# B&R Automation Studio project ControlPLC_DataDistribution (part 6)

#### vfAddAlarm.c
```c
#include <bur/plctypes.h>
#ifdef __cplusplus
	extern "C"
	{
#endif
	#include "VFAlarms.h"
#ifdef __cplusplus
	};
#endif
#include "string.h"

/* TODO: Add your comment here */
plcbit vfAddAlarm(plcstring* name, plcstring* scope, unsigned long code, enum vfALARMS_SEVERITY_enum severity, enum vfALARMS_BEHAVIOR_enum behavior, struct vfAlarms_Data_typ* data)
{

	vfAddAlarmTextScope( name, scope, "", code, severity, behavior, data);

	return 1;
}

plcbit vfAddAlarmApi(struct vfAlarms_Instance_type* name, plcstring* scope, unsigned long code, enum vfALARMS_SEVERITY_enum severity, enum vfALARMS_BEHAVIOR_enum behavior, struct vfAlarms_Data_typ* data){

	vfAddAlarm(name->_,  scope, code, severity, behavior, data);

	STRING snippet[vfALARMS_MAX_SNIPPET_PV_NAME_LEN];
	stringlcpy( snippet, data->in.snippetPvName, vfALARMS_MAX_SNIPPET_PV_NAME_LEN);
	stringlcat( snippet, ".", vfALARMS_MAX_SNIPPET_PV_NAME_LEN);
	stringlcat( snippet, name->snippet, vfALARMS_MAX_SNIPPET_PV_NAME_LEN);

	vfAddSnippet( name->snippet, snippet, data);

}

/* TODO: Add your comment here */
plcbit vfAddAlarmTextScope(plcstring* name, plcstring* scope, plcstring* textScope, unsigned long code, enum vfALARMS_SEVERITY_enum severity, enum vfALARMS_BEHAVIOR_enum behavior, struct vfAlarms_Data_typ* data)
{
	// Error check inputs.
	if (!data) return 0;
	if (!name) return 0;

	// Look for first empty spot, and add new alarm info there.
	int i;
	for (i = 0; i < vfALARMS_MAX_ALARMS; i++) {
		if (!strcmp(data->internal.alarms[i].name, "")) {
			// Found an empty location. Add our string.
			strcpy(data->internal.alarms[i].name, name);
			if (!strcmp(scope, "")) {
				strcpy(data->internal.alarms[i].scope, data->in.scope);
			} else {
				strcpy(data->internal.alarms[i].scope, scope);
			}

			if (!strcmp(textScope, "")) {
				strcpy(data->internal.alarms[i].textScope, data->in.scope);
			} else{
				strcpy(data->internal.alarms[i].textScope, textScope);
			}
			data->internal.alarms[i].code = code;
			data->internal.alarms[i].severity = severity;
			data->internal.alarms[i].behavior = behavior;
			break;
		}
	}

	return 1;
}

plcbit vfAddAlarmTextScopeApi(struct vfAlarms_Instance_type* name, plcstring* scope, plcstring* textScope, unsigned long code, enum vfALARMS_SEVERITY_enum severity, enum vfALARMS_BEHAVIOR_enum behavior, struct vfAlarms_Data_typ* data){

	vfAddAlarmTextScope(name->_,  scope, textScope, code, severity, behavior, data);

	STRING snippet[vfALARMS_MAX_SNIPPET_PV_NAME_LEN];
	stringlcpy( snippet, data->in.snippetPvName, vfALARMS_MAX_SNIPPET_PV_NAME_LEN);
	stringlcat( snippet, ".", vfALARMS_MAX_SNIPPET_PV_NAME_LEN);
	stringlcat( snippet, name->snippet, vfALARMS_MAX_SNIPPET_PV_NAME_LEN);

	vfAddSnippet( name->snippet, snippet, data);

}
```

#### vfAddSnippet.c
```c
#include <bur/plctypes.h>
#ifdef __cplusplus
	extern "C"
	{
#endif
	#include "VFAlarms.h"
#ifdef __cplusplus
	};
#endif
#include "string.h"

/* TODO: Add your comment here */
plcbit vfAddSnippet(plcstring* key, plcstring* pvName, struct vfAlarms_Data_typ* data)
{
	// Error check inputs.
	if (!data) return 0;
	if (!key) return 0;
	if (!pvName) return 0;

	// Look for first empty spot, and add new snippet info there.
	int i;
	for (i = 0; i < vfALARMS_MAX_SNIPPETS; i++) {
		if (!strcmp(data->internal.snippets[i].key, "")) {
			// Found an empty location. Add our string.
			strcpy(data->internal.snippets[i].key, key);
			strcpy(data->internal.snippets[i].pvName, pvName);
			break;
		}
	}

	return 1;
}
```

#### vfAddReactionByName.c
```c
#include <bur/plctypes.h>
#ifdef __cplusplus
	extern "C"
	{
#endif
	#include "VFAlarms.h"
#ifdef __cplusplus
	};
#endif
#include "string.h"

/* TODO: Add your comment here */
plcbit vfAddReactionByName(plcstring* name, plcstring* reactionName1, plcstring* reactionName2, plcstring* reactionName3, plcstring* reactionName4, plcstring* reactionName5, plcstring* reactionName6, struct vfAlarms_Data_typ* data)
{
	// Error check inputs.
	if (!data) return 0;
	if (!name) return 0;

	// Look for first empty spot, and add new alarm info there.
	int i;
	for (i = 0; i < vfALARMS_MAX_MAPPINGS; i++) {
		if (!strcmp(data->internal.reactions.byName[i].name, "")) {
			// Found an empty location. Add our info.
			strcpy(data->internal.reactions.byName[i].name, name);
			strcpy(data->internal.reactions.byName[i].reactionName[0], reactionName1);
			strcpy(data->internal.reactions.byName[i].reactionName[1], reactionName2);
			strcpy(data->internal.reactions.byName[i].reactionName[2], reactionName3);
			strcpy(data->internal.reactions.byName[i].reactionName[3], reactionName4);
			strcpy(data->internal.reactions.byName[i].reactionName[4], reactionName5);
			strcpy(data->internal.reactions.byName[i].reactionName[5], reactionName6);
			break;
		}
	}

	return 1;
}
```

#### vfAddReactionBySeverity.c
```c
#include <bur/plctypes.h>
#ifdef __cplusplus
	extern "C"
	{
#endif
	#include "VFAlarms.h"
#ifdef __cplusplus
	};
#endif
#include "string.h"

/* TODO: Add your comment here */
plcbit vfAddReactionBySeverity(enum vfALARMS_SEVERITY_enum severity, plcstring* reactionName1, plcstring* reactionName2, plcstring* reactionName3, plcstring* reactionName4, plcstring* reactionName5, plcstring* reactionName6, struct vfAlarms_Data_typ* data)
{
	// Error check inputs.
	if (!data) return 0;

	// Look for first empty spot, and add new alarm info there.
	int i;
	for (i = 0; i < vfALARMS_MAX_MAPPINGS; i++) {
		if (data->internal.reactions.bySeverity[i].severity == vfALARMS_SEVERITY_NONE) {
			// Found an empty location. Add our info.
			data->internal.reactions.bySeverity[i].severity = severity;
			strcpy(data->internal.reactions.bySeverity[i].reactionName[0], reactionName1);
			strcpy(data->internal.reactions.bySeverity[i].reactionName[1], reactionName2);
			strcpy(data->internal.reactions.bySeverity[i].reactionName[2], reactionName3);
			strcpy(data->internal.reactions.bySeverity[i].reactionName[3], reactionName4);
			strcpy(data->internal.reactions.bySeverity[i].reactionName[4], reactionName5);
			strcpy(data->internal.reactions.bySeverity[i].reactionName[5], reactionName6);
			break;
		}
	}

	return 1;
}
```

#### vfAddAggregationByName.c
```c
#include <bur/plctypes.h>
#ifdef __cplusplus
	extern "C"
	{
#endif
	#include "VFAlarms.h"
#ifdef __cplusplus
	};
#endif
#include "string.h"

/* TODO: Add your comment here */
plcbit vfAddAggregationByName(plcstring* name, plcstring* aggregationName, struct vfAlarms_Data_typ* data)
{
	// Error check inputs.
	if (!data) return 0;
	if (!name) return 0;

	// Look for first empty spot, and add new alarm info there.
	int i;
	for (i = 0; i < vfALARMS_MAX_MAPPINGS; i++) {
		if (!strcmp(data->internal.aggregations.byName[i].name, "")) {
			// Found an empty location. Add our info.
			strcpy(data->internal.aggregations.byName[i].name, name);
			strcpy(data->internal.aggregations.byName[i].aggregationName, aggregationName);
			break;
		}
	}

	return 1;
}

plcbit vfAddAggregationByNameApi(plcstring* name, struct vfAlarms_Instance_type* aggregationName, struct vfAlarms_Data_typ* data){

	vfAddAggregationByName( name, aggregationName->_, data);

}
```

#### vfAddAggregationBySeverity.c
```c
#include <bur/plctypes.h>
#ifdef __cplusplus
	extern "C"
	{
#endif
	#include "VFAlarms.h"
#ifdef __cplusplus
	};
#endif
#include "string.h"

/* TODO: Add your comment here */
plcbit vfAddAggregationBySeverity(enum vfALARMS_SEVERITY_enum severity, plcstring* aggregationName, struct vfAlarms_Data_typ* data)
{
	// Error check inputs.
	if (!data) return 0;

	// Look for first empty spot, and add new alarm info there.
	int i;
	for (i = 0; i < vfALARMS_MAX_MAPPINGS; i++) {
		if (data->internal.aggregations.bySeverity[i].severity == vfALARMS_SEVERITY_NONE) {
			// Found an empty location. Add our info.
			data->internal.aggregations.bySeverity[i].severity = severity;
			strcpy(data->internal.aggregations.bySeverity[i].aggregationName, aggregationName);
			break;
		}
	}

	return 1;
}
```

#### vfSetDefaultMapping.c
```c
#include <bur/plctypes.h>
#ifdef __cplusplus
	extern "C"
	{
#endif
	#include "VFAlarms.h"
#ifdef __cplusplus
	};
#endif
#include "string.h"

/* TODO: Add your comment here */
plcbit vfSetDefaultMapping(enum vfALARMS_MAPPING_enum type, plcstring* alarmName, struct vfAlarms_Data_typ* data)
{
	// Error check inputs.
	if (!data) return 0;

	data->internal.defaultMapping.type = type;
	strcpy(data->internal.defaultMapping.alarmName, alarmName);

	return 1;
}

plcbit vfSetDefaultMappingApi(enum vfALARMS_MAPPING_enum type, struct vfAlarms_Instance_type* alarmName, struct vfAlarms_Data_typ* data){

	vfSetDefaultMapping( type, alarmName->_ , data);

}
```

#### vfCreateAlarmsFaster.c
```c
#include <bur/plctypes.h>
#ifdef __cplusplus
	extern "C"
	{
#endif
	#include "VFAlarms.h"
#ifdef __cplusplus
	};
#endif

plcbit vfCreateAlarmsFaster(struct vfAlarms_Data_typ* data)
{
	// Error check inputs.
	if (!data) return 0;
	if (!data->in.mpLink) return 0;

	// Create the XML structure.
	buildXml(data, vfALARMS_XML_TYPE_START_WRITE);
	buildXml(data, vfALARMS_XML_TYPE_START_DOC);

	addXmlElement(data, "Configuration", 0);
		addXmlElement(data, "Version", 1, "ID", "1");
		closeXmlElement(data);
		addXmlElement(data, "Element", 1, "ID", data->in.mpLinkName);
			addXmlElement(data, "Group", 1, "ID", "mapp.AlarmX.Core");
				addXmlElement(data, "Group", 1, "ID", "Mapping");
					addMappingsByName(data);
				closeXmlElement(data);
				addXmlElement(data, "Group", 1, "ID", "BySeverity");
					addMappingsBySeverity(data);
				closeXmlElement(data);
				addXmlElement(data, "Group", 1, "ID", "Default");
					addDefaultMapping(data);
				closeXmlElement(data);
			closeXmlElement(data);
			// All user alarms get added here.
			addXmlElement(data, "Group", 1, "ID", "mapp.AlarmX.Core.Configuration");
				addAlarms(data);
			closeXmlElement(data);
			addXmlElement(data, "Group", 1, "ID", "mapp.AlarmX.Core.Categories");
				addCategories(data);
			closeXmlElement(data);
			addXmlElementFull(data, "Group", 1, "ID", "mapp.AlarmX.Core.Queries");
			addXmlElement(data, "Group", 1, "ID", "mapp.AlarmX.Core.Retain");
				addXmlElementFull(data, "Property", 3, "ID", "MemorySize", "DataType", "UDINT", "Value", "5");
				addXmlElementFull(data, "Property", 3, "ID", "MemoryType", "DataType", "DINT", "Value", "1");
			closeXmlElement(data);
			// All user defined snippets get added here.
			addXmlElement(data, "Group", 1, "ID", "mapp.AlarmX.Core.Snippets");
				addXmlElementFull(data, "Group", 1, "ID", "AutoDetect");
				addSnippets(data);
			closeXmlElement(data);
		closeXmlElement(data);
	closeXmlElement(data);

	buildXml(data, vfALARMS_XML_TYPE_END_DOC);
	buildXml(data, vfALARMS_XML_TYPE_GET_MEM);

	// Write the XML data to file.
	strcpy(data->internal.fileName, "config_");
	strcat(data->internal.fileName, data->in.scope);
	strcat(data->internal.fileName, ".xml");
	handleXmlFile(data, vfALARMS_FILE_CMD_DELETE);
	handleXmlFile(data, vfALARMS_FILE_CMD_SAVE);

	// Create the Mapp configuration object on the target based on the XML file.
	createMappConfig(data);

	// Close the XML writer (which wipes out our data buffer).
	buildXml(data, vfALARMS_XML_TYPE_END_WRITE);

	data->out.done = !data->out.error;

}

void addDefaultMapping(struct vfAlarms_Data_typ* data) {

	switch(data->internal.defaultMapping.type) {
		case vfALARMS_MAPPING_REMAIN:
			addXmlElement(data, "Group", 1, "ID", "[0]");
				addXmlElementFull(data, "Property", 3, "ID", "Type", "DataType", "STRING", "Value", "Remain");
			closeXmlElement(data);
			break;

		case vfALARMS_MAPPING_AGGREGATE:
			addXmlElement(data, "Group", 1, "ID", "[0]");
				addXmlElementFull(data, "Property", 3, "ID", "Type", "DataType", "STRING", "Value", "Aggregate");
				addXmlElementFull(data, "Property", 3, "ID", "Name", "DataType", "STRING", "Value", data->internal.defaultMapping.alarmName);
			closeXmlElement(data);
			break;

		case vfALARMS_MAPPING_ESCALATE:
			addXmlElement(data, "Group", 1, "ID", "[0]");
				addXmlElementFull(data, "Property", 3, "ID", "Type", "DataType", "STRING", "Value", "Escalate Alarm");
			closeXmlElement(data);
			break;
	}
}

void addMappingsByName(struct vfAlarms_Data_typ* data) {

	int i = 0;
	int j = 0;
	STRING * tempString[80];
	STRING * index[10];
	int storedIndex = 0;

	// Loop through all reaction mappings by name.
	for (i = 0; i < vfALARMS_MAX_MAPPINGS; i++) {

		if (strcmp(data->internal.reactions.byName[i].name, "")) {

			// Create the dynamic index.
			brsitoa(storedIndex, tempString);
			strcpy(index, "[");
			strcat(index, tempString);
			strcat(index, "]");

			addXmlElement(data, "Group", 1, "ID", index);
			addXmlElementFull(data, "Property", 3, "ID", "Alarm", "DataType", "STRING", "Value", data->internal.reactions.byName[i].name);
			for (j = 0; j <= vfALARMS_MAI_REACTIONS; j++) {
				if (strcmp(data->internal.reactions.byName[i].reactionName[j], "")) {
					brsitoa(j, tempString);
					strcpy(index, "[");
					strcat(index, tempString);
					strcat(index, "]");
					addXmlElement(data, "Group", 1, "ID", index);
					//	addXmlElementFull(data, "Property", 3, "ID", "Name", "DataType", "STRING", "Value", data->internal.reactions.byName[i].reactionName[j]);
					//	addXmlElementFull(data, "Property", 3, "ID", "Type", "DataType", "STRING", "Value", "Reaction");

					//Modified by Paul to Escalate Reactions
					addXmlElementFull(data, "Property", 3, "ID", "Reaction", "DataType", "STRING", "Value", data->internal.reactions.byName[i].reactionName[j]);
					addXmlElementFull(data, "Property", 3, "ID", "Type", "DataType", "STRING", "Value", "EscalateReaction");

					closeXmlElement(data);
				}
			}
			closeXmlElement(data);
			storedIndex++;
		}

		if (strcmp(data->internal.reactions.byNameNotEscalated[i].name, "")) {
			// Create the dynamic index.
			brsitoa(storedIndex, tempString);
			strcpy(index, "[");
			strcat(index, tempString);
			strcat(index, "]");

			addXmlElement(data, "Group", 1, "ID", index);
			addXmlElementFull(data, "Property", 3, "ID", "Alarm", "DataType", "STRING", "Value", data->internal.reactions.byNameNotEscalated[i].name);
			for (j = 0; j <= vfALARMS_MAI_REACTIONS; j++) {
				if (strcmp(data->internal.reactions.byNameNotEscalated[i].reactionName[j], "")) {
					brsitoa(j, tempString);
					strcpy(index, "[");
					strcat(index, tempString);
					strcat(index, "]");
					addXmlElement(data, "Group", 1, "ID", index);
						addXmlElementFull(data, "Property", 3, "ID", "Name", "DataType", "STRING", "Value", data->internal.reactions.byNameNotEscalated[i].reactionName[j]);
						addXmlElementFull(data, "Property", 3, "ID", "Type", "DataType", "STRING", "Value", "Reaction");

					//Modified by Paul to Escalate Reactions
					//	addXmlElementFull(data, "Property", 3, "ID", "Reaction", "DataType", "STRING", "Value", data->internal.reactions.byName[i].reactionName[j]);
					//	addXmlElementFull(data, "Property", 3, "ID", "Type", "DataType", "STRING", "Value", "EscalateReaction");

					closeXmlElement(data);
				}
			}
			closeXmlElement(data);
			storedIndex++;
		}
	}

	// Loop through all aggregation mappings by name.
	for (i = 0; i < vfALARMS_MAX_MAPPINGS; i++) {
		if (strcmp(data->internal.aggregations.byName[i].name, "")) {
			// Create the dynamic index.
			brsitoa(storedIndex, tempString);
			strcpy(index, "[");
			strcat(index, tempString);
			strcat(index, "]");

			addXmlElement(data, "Group", 1, "ID", index);
				addXmlElementFull(data, "Property", 3, "ID", "Alarm", "DataType", "STRING", "Value", data->internal.aggregations.byName[i].name);
				addXmlElement(data, "Group", 1, "ID", "[0]");
					addXmlElementFull(data, "Property", 3, "ID", "Name", "DataType", "STRING", "Value", data->internal.aggregations.byName[i].aggregationName);
					addXmlElementFull(data, "Property", 3, "ID", "Type", "DataType", "STRING", "Value", "Aggregate");
				closeXmlElement(data);
			closeXmlElement(data);
			storedIndex++;
		}
	}

	if( data->in.escalateAll ){
		// Create the dynamic index.
		brsitoa(storedIndex, tempString);
		strcpy(index, "[");
		strcat(index, tempString);
		strcat(index, "]");

		addXmlElement(data, "Group", 1, "ID", index);
			addXmlElementFull(data, "Property", 3, "ID", "Alarm", "DataType", "STRING", "Value", "*");
			addXmlElement(data, "Group", 1, "ID", "[0]");
				addXmlElementFull(data, "Property", 3, "ID", "Type", "DataType", "STRING", "Value", "Escalate");
			closeXmlElement(data);
		closeXmlElement(data);
		storedIndex++;
	}
}

void addMappingsBySeverity(struct vfAlarms_Data_typ* data) {

	int i = 0;
	int j = 0;
	STRING * tempString[80];
	STRING * index[10];
	STRING * severity[80];
	int storedIndex = 0;

	// Loop through all reaction mappings by severity.
	for (i = 0; i < vfALARMS_MAX_MAPPINGS; i++) {
		if (data->internal.reactions.bySeverity[i].severity != vfALARMS_SEVERITY_NONE) {
			storedIndex = i;

			// Create the dynamic index.
			brsitoa(i, tempString);
			strcpy(index, "[");
			strcat(index, tempString);
			strcat(index, "]");

			// Create the 'severity' string field.
			brsitoa(data->internal.reactions.bySeverity[i].severity, severity);

			addXmlElement(data, "Group", 1, "ID", index);
				addXmlElementFull(data, "Property", 3, "ID", "Severity", "DataType", "STRING", "Value", severity);
				for (j = 0; j <= vfALARMS_MAI_REACTIONS; j++) {
					if (strcmp(data->internal.reactions.bySeverity[i].reactionName[j], "")) {
						brsitoa(j, tempString);
						strcpy(index, "[");
						strcat(index, tempString);
						strcat(index, "]");
						addXmlElement(data, "Group", 1, "ID", index);
							addXmlElementFull(data, "Property", 3, "ID", "Name", "DataType", "STRING", "Value", data->internal.reactions.bySeverity[i].reactionName[j]);
							addXmlElementFull(data, "Property", 3, "ID", "Type", "DataType", "STRING", "Value", "Reaction");

						closeXmlElement(data);
					}
				}
			closeXmlElement(data);
		}
	}

	// Loop through all aggregation mappings by severity
	for (i = 0; i < vfALARMS_MAX_MAPPINGS; i++) {
		if (data->internal.aggregations.bySeverity[i].severity != vfALARMS_SEVERITY_NONE) {

			// Create the dynamic index.
			brsitoa(i+storedIndex, tempString);
			strcpy(index, "[");
			strcat(index, tempString);
			strcat(index, "]");

			// Create the 'severity' string field.
			brsitoa(data->internal.aggregations.bySeverity[i].severity, severity);

			addXmlElement(data, "Group", 1, "ID", index);
				addXmlElementFull(data, "Property", 3, "ID", "Severity", "DataType", "STRING", "Value", severity);
				addXmlElement(data, "Group", 1, "ID", "[0]");
					addXmlElementFull(data, "Property", 3, "ID", "Name", "DataType", "STRING", "Value", data->internal.aggregations.bySeverity[i].aggregationName);
					addXmlElementFull(data, "Property", 3, "ID", "Type", "DataType", "STRING", "Value", "Aggregate");
				closeXmlElement(data);
			closeXmlElement(data);
		}
	}
}

void addAlarms(struct vfAlarms_Data_typ* data) {

	int i = 0;
	STRING * tempString[80];
	STRING * index[10];
	STRING * severity[80];
	STRING * code[80];
	STRING * message[255];
	STRING * additionalInfo1[255];
	STRING * additionalInfo2[255];
	for (i = 0; i < vfALARMS_MAX_ALARMS; i++) {
		if (strcmp(data->internal.alarms[i].name, "")) {

			// Create the dynamic index.
			brsitoa(i, tempString);
			strcpy(index, "[");
			strcat(index, tempString);
			strcat(index, "]");

			// Create the 'severity' string field.
			brsitoa(data->internal.alarms[i].severity, severity);

			// Create the 'code' string field.
			brsitoa(data->internal.alarms[i].code, code);

			// Create the 'message' string field.
			strcpy(message, "{$IAT/");
			strcat(message, data->internal.alarms[i].textScope);
			strcat(message, "/");
			strcat(message, data->internal.alarms[i].name);
			strcat(message, ".Message}");

			// Create the 'additionalInfo' string field.
			strcpy(additionalInfo1, "{$IAT/");
			strcat(additionalInfo1, data->internal.alarms[i].textScope);
			strcat(additionalInfo1, "/");
			strcat(additionalInfo1, data->internal.alarms[i].name);
			strcat(additionalInfo1, ".AdditionalInfo}");

			// Create the 'additionalInfo2' string field.
			// This is being used to store the scope of the alarm, actually.
			strcpy(additionalInfo2, data->internal.alarms[i].scope);

			addXmlElement(data, "Group", 1, "ID", index);
				addXmlElementFull(data, "Property", 3, "ID", "Name", "DataType", "STRING", "Value", data->internal.alarms[i].name);
				addXmlElementFull(data, "Property", 3, "ID", "Message", "DataType", "STRING", "Value", message);
				addXmlElementFull(data, "Property", 3, "ID", "Code", "DataType", "UDINT", "Value", code);
				addXmlElementFull(data, "Property", 3, "ID", "Severity", "DataType", "UDINT", "Value", severity);
				addXmlElementFull(data, "Property", 3, "ID", "AdditionalInformation1", "DataType", "STRING", "Value", additionalInfo1);
				addXmlElementFull(data, "Property", 3, "ID", "AdditionalInformation2", "DataType", "STRING", "Value", additionalInfo2);
				addXmlElementFull(data, "Property", 3, "ID", "Disable", "DataType", "BOOL", "Value", "false");
				addXmlElement(data, "Group", 1, "ID", "Behavior");
					addAlarmBehavior(data, i);
				closeXmlElement(data);
			closeXmlElement(data);

		}
	}
}

void addCategories(struct vfAlarms_Data_typ* data) {

	addXmlElement(data, "Group", 1, "ID", "[0]");
		addXmlElementFull(data, "Property", 3, "ID", "Name", "DataType", "STRING", "Value", "Information");
		addXmlElement(data, "Group", 1, "ID", "SourceProperty");
			addXmlElementFull(data, "Property", 3, "ID", "Severity", "DataType", "STRING", "Value", "1");
		closeXmlElement(data);
	closeXmlElement(data);
	addXmlElement(data, "Group", 1, "ID", "[1]");
		addXmlElementFull(data, "Property", 3, "ID", "Name", "DataType", "STRING", "Value", "Warning");
		addXmlElement(data, "Group", 1, "ID", "SourceProperty");
			addXmlElementFull(data, "Property", 3, "ID", "Severity", "DataType", "STRING", "Value", "2");
		closeXmlElement(data);
	closeXmlElement(data);
	addXmlElement(data, "Group", 1, "ID", "[2]");
		addXmlElementFull(data, "Property", 3, "ID", "Name", "DataType", "STRING", "Value", "Alarm");
		addXmlElement(data, "Group", 1, "ID", "SourceProperty");
			addXmlElementFull(data, "Property", 3, "ID", "Severity", "DataType", "STRING", "Value", "3");
		closeXmlElement(data);
	closeXmlElement(data);
	addXmlElement(data, "Group", 1, "ID", "[3]");
		addXmlElementFull(data, "Property", 3, "ID", "Name", "DataType", "STRING", "Value", "Critical");
		addXmlElement(data, "Group", 1, "ID", "SourceProperty");
			addXmlElementFull(data, "Property", 3, "ID", "Severity", "DataType", "STRING", "Value", "4");
		closeXmlElement(data);
	closeXmlElement(data);

}

void addAlarmBehavior(struct vfAlarms_Data_typ* data, UINT i) {

	switch(data->internal.alarms[i].behavior) {
		case vfALARMS_BEHAVIOR_EDGE:
			addXmlElementFull(data, "Property", 3, "ID", "Acknowledge", "DataType", "DINT", "Value", "1");
			addXmlElementFull(data, "Property", 3, "ID", "AutoReset", "DataType", "BOOL", "Value", "true");
			addXmlElementFull(data, "Property", 3, "ID", "MultipleInstances", "DataType", "BOOL", "Value", "true");
			addXmlElementFull(data, "Property", 3, "ID", "ReactionUntilAcknowledged", "DataType", "BOOL", "Value", "true");
			addXmlElementFull(data, "Property", 3, "ID", "Retain", "DataType", "BOOL", "Value", "false");
			addXmlElementFull(data, "Property", 3, "ID", "Type", "DataType", "STRING", "Value", "EdgeAlarm");
			addXmlElement(data, "Group", 1, "ID", "DataUpdate");
				addXmlElement(data, "Group", 1, "ID", "Activation");
					addXmlElementFull(data, "Property", 3, "ID", "Snippets", "DataType", "BOOL", "Value", "false");
					addXmlElementFull(data, "Property", 3, "ID", "TimeStamp", "DataType", "BOOL", "Value", "false");
				closeXmlElement(data);
			closeXmlElement(data);
			addXmlElement(data, "Group", 1, "ID", "Recording");
				addXmlElementFull(data, "Property", 3, "ID", "AcknowledgedToUnacknowledged", "DataType", "BOOL", "Value", "false");
				addXmlElementFull(data, "Property", 3, "ID", "ActiveToInactive", "DataType", "BOOL", "Value", "false");
				addXmlElementFull(data, "Property", 3, "ID", "InactiveToActive", "DataType", "BOOL", "Value", "true");
				addXmlElementFull(data, "Property", 3, "ID", "UnacknowledgedToAcknowledged", "DataType", "BOOL", "Value", "true");
			closeXmlElement(data);
			break;

		case vfALARMS_BEHAVIOR_PERSISTENT:
			addXmlElementFull(data, "Property", 3, "ID", "Acknowledge", "DataType", "DINT", "Value", "1");
			addXmlElementFull(data, "Property", 3, "ID", "AutoReset", "DataType", "BOOL", "Value", "false");
			addXmlElementFull(data, "Property", 3, "ID", "MultipleInstances", "DataType", "BOOL", "Value", "false");
			addXmlElementFull(data, "Property", 3, "ID", "ReactionUntilAcknowledged", "DataType", "BOOL", "Value", "true");
			addXmlElementFull(data, "Property", 3, "ID", "Retain", "DataType", "BOOL", "Value", "false");
			addXmlElementFull(data, "Property", 3, "ID", "Type", "DataType", "STRING", "Value", "PersistentAlarm");
			addXmlElement(data, "Group", 1, "ID", "DataUpdate");
				addXmlElement(data, "Group", 1, "ID", "Activation");
					addXmlElementFull(data, "Property", 3, "ID", "Snippets", "DataType", "BOOL", "Value", "false");
					addXmlElementFull(data, "Property", 3, "ID", "TimeStamp", "DataType", "BOOL", "Value", "false");
				closeXmlElement(data);
			closeXmlElement(data);
			addXmlElement(data, "Group", 1, "ID", "Recording");
				addXmlElementFull(data, "Property", 3, "ID", "AcknowledgedToUnacknowledged", "DataType", "BOOL", "Value", "true");
				addXmlElementFull(data, "Property", 3, "ID", "ActiveToInactive", "DataType", "BOOL", "Value", "false");
				addXmlElementFull(data, "Property", 3, "ID", "InactiveToActive", "DataType", "BOOL", "Value", "true");
				addXmlElementFull(data, "Property", 3, "ID", "UnacknowledgedToAcknowledged", "DataType", "BOOL", "Value", "true");
				addXmlElementFull(data, "Property", 3, "ID", "Update", "DataType", "BOOL", "Value", "false");
			closeXmlElement(data);
			break;

	}
}

void addSnippets(struct vfAlarms_Data_typ* data) {

	int i = 0;
	STRING * tempString[80];
	STRING * index[10];
	for (i = 0; i < vfALARMS_MAX_SNIPPETS; i++) {
		if (strcmp(data->internal.snippets[i].key, "")) {

			// Create the dynamic index.
			brsitoa(i, tempString);
			strcpy(index, "[");
			strcat(index, tempString);
			strcat(index, "]");

			addXmlElement(data, "Group", 1, "ID", index);
				addXmlElementFull(data, "Property", 3, "ID", "Alarm", "DataType", "STRING", "Value", "");
				addXmlElementFull(data, "Property", 3, "ID", "Key", "DataType", "STRING", "Value", data->internal.snippets[i].key);
				addXmlElement(data, "Group", 1, "ID", "Value");
					addXmlElementFull(data, "Property", 3, "ID", "PV", "DataType", "STRING", "Value", data->internal.snippets[i].pvName);
					addXmlElementFull(data, "Property", 3, "ID", "Type", "DataType", "DINT", "Value", "1");
				closeXmlElement(data);
			closeXmlElement(data);

		}
	}
}

void addXmlElementFull(struct vfAlarms_Data_typ* data, plcstring* name, USINT numAttributes, plcstring* attribute1, plcstring* value1, plcstring* attribute2, plcstring* value2, plcstring* attribute3, plcstring* value3) {
	addXmlElement(data, name, numAttributes, attribute1, value1, attribute2, value2, attribute3, value3);
	buildXml(data, vfALARMS_XML_TYPE_END_ELEM);
}

void addXmlElement(struct vfAlarms_Data_typ* data, plcstring* name, USINT numAttributes, plcstring* attribute1, plcstring* value1, plcstring* attribute2, plcstring* value2, plcstring* attribute3, plcstring* value3) {
	buildXml(data, vfALARMS_XML_TYPE_START_ELEM, name);
	if (numAttributes > 0) {
		buildXml(data, vfALARMS_XML_TYPE_ATTRIBUTE, attribute1, value1);
	}
	if (numAttributes > 1) {
		buildXml(data, vfALARMS_XML_TYPE_ATTRIBUTE, attribute2, value2);
	}
	if (numAttributes > 2) {
		buildXml(data, vfALARMS_XML_TYPE_ATTRIBUTE, attribute3, value3);
	}
}

void closeXmlElement(struct vfAlarms_Data_typ* data) {
	buildXml(data, vfALARMS_XML_TYPE_END_ELEM);
}

void buildXml(struct vfAlarms_Data_typ* data, enum vfALARMS_XML_TYPE_enum type, plcstring* arg1, plcstring* arg2, plcstring* arg3) {

	// Skip the step if there's an active error.
	if (data->out.error) return;

	BOOL done = 0;
	BOOL error = 0;
	UINT errorId = 0;
	STRING errorString[80];
	strcpy(errorString, "");
	while (!done && !error) {

		// Call all FUBs so we get the initial 65534 status.
		xmlCreateMemoryWriter(&data->internal.fub.xmlCreateMemoryWriter);
		xmlWriteStartDocument(&data->internal.fub.xmlWriteStartDocument);
		xmlWriteStartElement(&data->internal.fub.xmlWriteStartElement);
		xmlWriteAttribute(&data->internal.fub.xmlWriteAttribute);
		xmlWriteEndElement(&data->internal.fub.xmlWriteEndElement);
		xmlWriteEndDocument(&data->internal.fub.xmlWriteEndDocument);
		xmlGetMemoryInfo(&data->internal.fub.xmlGetMemoryInfo);
		xmlCloseMemoryWriter(&data->internal.fub.xmlCloseMemoryWriter);
		data->internal.fub.xmlCreateMemoryWriter.enable = 0;
		data->internal.fub.xmlWriteStartDocument.enable = 0;
		data->internal.fub.xmlWriteStartElement.enable = 0;
		data->internal.fub.xmlWriteAttribute.enable = 0;
		data->internal.fub.xmlWriteEndElement.enable = 0;
		data->internal.fub.xmlWriteEndDocument.enable = 0;
		data->internal.fub.xmlGetMemoryInfo.enable = 0;
		data->internal.fub.xmlCloseMemoryWriter.enable = 0;

		switch(type) {
			case vfALARMS_XML_TYPE_START_WRITE:
				if (data->internal.fub.xmlCreateMemoryWriter.status == ERR_OK) {
					data->internal.xmlIdent = data->internal.fub.xmlCreateMemoryWriter.ident;
					done = 1;
				} else if ((data->internal.fub.xmlCreateMemoryWriter.status != ERR_FUB_ENABLE_FALSE) && (data->internal.fub.xmlCreateMemoryWriter.status != ERR_FUB_BUSY)) {
					error = 1;
					errorId = data->internal.fub.xmlCreateMemoryWriter.status;
					strcpy(errorString, "Error while creating the memory writer");
				} else {
					data->internal.fub.xmlCreateMemoryWriter.enable = 1;
				}
				break;

			case vfALARMS_XML_TYPE_START_DOC:
				if (data->internal.fub.xmlWriteStartDocument.status == ERR_OK) {
					done = 1;
				} else if ((data->internal.fub.xmlWriteStartDocument.status != ERR_FUB_ENABLE_FALSE) && (data->internal.fub.xmlWriteStartDocument.status != ERR_FUB_BUSY)) {
					error = 1;
					errorId = data->internal.fub.xmlWriteStartDocument.status;
					strcpy(errorString, "Error while writing start document");
				} else {
					data->internal.fub.xmlWriteStartDocument.enable = 1;
					data->internal.fub.xmlWriteStartDocument.ident = data->internal.xmlIdent;
					data->internal.fub.xmlWriteStartDocument.pVersion = &"1.0";
					data->internal.fub.xmlWriteStartDocument.pEncoding = &"UTF-8";
				}
				break;

			case vfALARMS_XML_TYPE_START_ELEM:
				if (data->internal.fub.xmlWriteStartElement.status == ERR_OK) {
					done = 1;
				} else if ((data->internal.fub.xmlWriteStartElement.status != ERR_FUB_ENABLE_FALSE) && (data->internal.fub.xmlWriteStartElement.status != ERR_FUB_BUSY)) {
					error = 1;
					errorId = data->internal.fub.xmlWriteStartElement.status;
					strcpy(errorString, "Error while writing start element");
				} else {
					data->internal.fub.xmlWriteStartElement.enable = 1;
					data->internal.fub.xmlWriteStartElement.ident = data->internal.xmlIdent;
					data->internal.fub.xmlWriteStartElement.pName = arg1;
				}
				break;

			case vfALARMS_XML_TYPE_ATTRIBUTE:
				if (data->internal.fub.xmlWriteAttribute.status == ERR_OK) {
					done = 1;
				} else if ((data->internal.fub.xmlWriteAttribute.status != ERR_FUB_ENABLE_FALSE) && (data->internal.fub.xmlWriteAttribute.status != ERR_FUB_BUSY)) {
					error = 1;
					errorId = data->internal.fub.xmlWriteAttribute.status;
					strcpy(errorString, "Error while writing attribute");
				} else {
					data->internal.fub.xmlWriteAttribute.enable = 1;
					data->internal.fub.xmlWriteAttribute.ident = data->internal.xmlIdent;
					data->internal.fub.xmlWriteAttribute.pName = arg1;
					data->internal.fub.xmlWriteAttribute.pValue = arg2;
				}
				break;

			case vfALARMS_XML_TYPE_END_ELEM:
				if (data->internal.fub.xmlWriteEndElement.status == ERR_OK) {
					done = 1;
				} else if ((data->internal.fub.xmlWriteEndElement.status != ERR_FUB_ENABLE_FALSE) && (data->internal.fub.xmlWriteEndElement.status != ERR_FUB_BUSY)) {
					error = 1;
					errorId = data->internal.fub.xmlWriteEndElement.status;
					strcpy(errorString, "Error while writing end element");
				} else {
					data->internal.fub.xmlWriteEndElement.enable = 1;
					data->internal.fub.xmlWriteEndElement.ident = data->internal.xmlIdent;
				}
				break;

			case vfALARMS_XML_TYPE_END_DOC:
				if (data->internal.fub.xmlWriteEndDocument.status == ERR_OK) {
					done = 1;
				} else if ((data->internal.fub.xmlWriteEndDocument.status != ERR_FUB_ENABLE_FALSE) && (data->internal.fub.xmlWriteEndDocument.status != ERR_FUB_BUSY)) {
					error = 1;
					errorId = data->internal.fub.xmlWriteEndDocument.status;
					strcpy(errorString, "Error while writing end document");
				} else {
					data->internal.fub.xmlWriteEndDocument.enable = 1;
					data->internal.fub.xmlWriteEndDocument.ident = data->internal.xmlIdent;
				}
				break;

			case vfALARMS_XML_TYPE_GET_MEM:
				if (data->internal.fub.xmlGetMemoryInfo.status == ERR_OK) {
					if (data->internal.fub.xmlGetMemoryInfo.xmlDataSize < vfALARMS_MAI_BUFFER) {
						data->internal.pXmlData = data->internal.fub.xmlGetMemoryInfo.pXmlData;
						data->internal.szXmlData = data->internal.fub.xmlGetMemoryInfo.xmlDataSize;
						done = 1;
					} else {
						error = 1;
						errorId = 50001;
					}
				} else if ((data->internal.fub.xmlGetMemoryInfo.status != ERR_FUB_ENABLE_FALSE) && (data->internal.fub.xmlGetMemoryInfo.status != ERR_FUB_BUSY)) {
					error = 1;
					errorId = data->internal.fub.xmlGetMemoryInfo.status;
					strcpy(errorString, "Error while retrieving mem info");
				} else {
					data->internal.fub.xmlGetMemoryInfo.enable = 1;
					data->internal.fub.xmlGetMemoryInfo.ident = data->internal.xmlIdent;
				}
				break;

			case vfALARMS_XML_TYPE_END_WRITE:
				if (data->internal.fub.xmlCloseMemoryWriter.status == ERR_OK) {
					done = 1;
				} else if ((data->internal.fub.xmlCloseMemoryWriter.status != ERR_FUB_ENABLE_FALSE) && (data->internal.fub.xmlCloseMemoryWriter.status != ERR_FUB_BUSY)) {
					error = 1;
					errorId = data->internal.fub.xmlCloseMemoryWriter.status;
					strcpy(errorString, "Error while closing the memory writer");
				} else {
					data->internal.fub.xmlCloseMemoryWriter.enable = 1;
					data->internal.fub.xmlCloseMemoryWriter.ident = data->internal.xmlIdent;
				}
				break;

			default:
				break;
		}
	}

	data->out.error = error;
	data->out.errorId = (DINT)errorId;
	strcpy(data->out.errorString, errorString);
}

void handleXmlFile(struct vfAlarms_Data_typ* data, enum vfALARMS_FILE_CMD_enum cmd) {

	// Skip the step if there's an active error.
	if (data->out.error) return;

	BOOL done = 0;
	BOOL error = 0;
	UINT errorId = 0;
	STRING errorString[80];
	strcpy(errorString, "");
	while (!done && !error) {

		FIOWrapFn_Cyclic(&data->internal.fub.fioWrapper);
		data->internal.fub.fioWrapper.IN.CMD.SaveAs = 0;
		data->internal.fub.fioWrapper.IN.CMD.Delete = 0;

		switch(cmd) {
			case vfALARMS_FILE_CMD_DELETE:
				if (data->internal.fub.fioWrapper.OUT.STAT.Done) {
					done = 1;
				} else if (data->internal.fub.fioWrapper.OUT.STAT.Error) {
					error = 1;
					errorId = data->internal.fub.fioWrapper.OUT.STAT.ErrorID;
					strcpy(errorString, "Error while deleting XML file");
				} else {
					data->internal.fub.fioWrapper.IN.CMD.Delete = 1;
					strcpy(data->internal.fub.fioWrapper.IN.PAR.FileDevice, data->in.deviceName);
					strcpy(data->internal.fub.fioWrapper.IN.PAR.FileName, data->internal.fileName);
				}
				break;

			case vfALARMS_FILE_CMD_SAVE:
				if (data->internal.fub.fioWrapper.OUT.STAT.Done) {
					done = 1;
				} else if (data->internal.fub.fioWrapper.OUT.STAT.Error) {
					error = 1;
					errorId = data->internal.fub.fioWrapper.OUT.STAT.ErrorID;
					strcpy(errorString, "Error while creating XML file");
				} else {
					data->internal.fub.fioWrapper.IN.CMD.SaveAs = 1;
					strcpy(data->internal.fub.fioWrapper.IN.PAR.FileDevice, data->in.deviceName);
					strcpy(data->internal.fub.fioWrapper.IN.PAR.FileName, data->internal.fileName);
					data->internal.fub.fioWrapper.IN.PAR.pData = data->internal.pXmlData;
					data->internal.fub.fioWrapper.IN.PAR.len = data->internal.szXmlData;
					data->internal.fub.fioWrapper.IN.PAR.offset = 0;
				}
				break;
		}
	}
	data->out.error = error;
	data->out.errorId = (DINT)errorId;
	strcpy(data->out.errorString, errorString);
}

void createMappConfig(struct vfAlarms_Data_typ* data) {

	// Skip the step if there's an active error.
	if (data->out.error) return;

	BOOL done = 0;
	BOOL error = 0;
	UINT errorId = 0;
	STRING errorString[80];
	strcpy(errorString, "");
	while (!done && !error) {

		MpComConfigManager(&data->internal.fub.manageConfiguration);
		data->internal.fub.manageConfiguration.Export = 0;
		data->internal.fub.manageConfiguration.Import = 0;

		data->internal.fub.manageConfiguration.Enable = 1;

		if (data->internal.fub.manageConfiguration.Active) {
			if (data->internal.fub.manageConfiguration.CommandBusy) {
//				data->internal.fub.manageConfiguration.Export = 1;
			} else if (data->internal.fub.manageConfiguration.Error) {
				error = 1;
				errorId = data->internal.fub.manageConfiguration.StatusID;
				strcpy(errorString, "Error while creating Mapp configuration");
			} else if (data->internal.fub.manageConfiguration.CommandDone) {
				done = 1;
			} else {
				data->internal.fub.manageConfiguration.DeviceName = &data->in.deviceName;
				data->internal.fub.manageConfiguration.FileName = &data->internal.fileName;
				data->internal.fub.manageConfiguration.MpLink = data->in.mpLink;
				data->internal.fub.manageConfiguration.Scope = mpCOM_CONFIG_SCOPE_COMPONENT;
				data->internal.fub.manageConfiguration.Import = 1;
			}
		}
	}
	data->out.error = error;
	data->out.errorId = (DINT)errorId;
	strcpy(data->out.errorString, errorString);
}
```

#### vfAddLogOriginMapping.c
```c
#include <bur/plctypes.h>
#ifdef __cplusplus
	extern "C"
	{
#endif
	#include "VFAlarms.h"
#ifdef __cplusplus
	};
#endif
#include "string.h"

/* TODO: Add your comment here */
plcbit vfAddLogOriginMapping(plcstring* originRaw, plcstring* originFormatted, struct Log_Origin_Mappings_typ* map)
{
	if (!map) return;

	int i = 0;

	// Search for first open spot for adding mappings.
	for (i = 0; i <= LOGBOOK_MAI_MAPPINGS; i++) {
		if (!strcmp(map->originRaw[i], "")) {
			strcpy(map->originRaw[i], originRaw);
			strcpy(map->originFormatted[i], originFormatted);
			return;
		}
	}
}
```

#### vfLookupOrigin.c
```c
#include <bur/plctypes.h>
#ifdef __cplusplus
	extern "C"
	{
#endif
	#include "VFAlarms.h"
#ifdef __cplusplus
	};
#endif
#include "string.h"

/* TODO: Add your comment here */
plcbit vfLookupOrigin(unsigned long pOriginRaw, unsigned long pOriginFormatted, struct Log_Origin_Mappings_typ* map)
{
	if (!map) return;

	int i = 0;

	char *originRaw = (char *)pOriginRaw;
	char *originFormatted = (char *)pOriginFormatted;

	// Loop through map, looking for a match.
	for (i = 0; i <= LOGBOOK_MAI_MAPPINGS; i++) {
		if (!strcmp(originRaw, map->originRaw[i])) {
			strcpy(originFormatted, map->originFormatted[i]);
			return;
		}
	}

	// Getting here means no match was found. Just pass the input back out.
	strcpy(originFormatted, originRaw);
}
```

#### vfAddNonEscalatedReactionByName.c
```c
#include <bur/plctypes.h>
#ifdef __cplusplus
	extern "C"
	{
#endif
	#include "VFAlarms.h"
#ifdef __cplusplus
	};
#endif
#include "string.h"

/* TODO: Add your comment here */
plcbit vfAddNonEscalatedReactionByName(plcstring* name, plcstring* reactionName1, plcstring* reactionName2, plcstring* reactionName3, plcstring* reactionName4, plcstring* reactionName5, plcstring* reactionName6, struct vfAlarms_Data_typ* data)
{
	// Error check inputs.
	if (!data) return 0;
	if (!name) return 0;

	// Look for first empty spot, and add new alarm info there.
	int i;
	for (i = 0; i < vfALARMS_MAX_MAPPINGS; i++) {
		if (!strcmp(data->internal.reactions.byName[i].name, "")) {
			// Found an empty location. Add our info.
			strcpy(data->internal.reactions.byNameNotEscalated[i].name, name);
			strcpy(data->internal.reactions.byNameNotEscalated[i].reactionName[0], reactionName1);
			strcpy(data->internal.reactions.byNameNotEscalated[i].reactionName[1], reactionName2);
			strcpy(data->internal.reactions.byNameNotEscalated[i].reactionName[2], reactionName3);
			strcpy(data->internal.reactions.byNameNotEscalated[i].reactionName[3], reactionName4);
			strcpy(data->internal.reactions.byNameNotEscalated[i].reactionName[4], reactionName5);
			strcpy(data->internal.reactions.byNameNotEscalated[i].reactionName[5], reactionName6);
			break;
		}
	}

	return 1;
}
```

#### vfAlarmEdge.c
```c
#include <bur/plctypes.h>
#ifdef __cplusplus
	extern "C"
	{
#endif
	#include "VFAlarms.h"
#ifdef __cplusplus
	};
#endif

plcbit vfAlarmEdge(struct vfAlarms_Component_typ* alarmComponent, struct vfAlarms_Instance_type* alarm){

	MpAlarmXSet( &alarmComponent->link, alarm->_);

}
plcbit vfAlarmEdgeSnippet(struct vfAlarms_Component_typ* alarmComponent, struct vfAlarms_Instance_type* alarm, plcstring* snippet){

	strncpy(alarm->snippet, snippet, sizeof(alarm->snippet) );

	vfAlarmEdge( alarmComponent, alarm );

}
```

#### vfAlarmPersistent.c
```c
#include <bur/plctypes.h>
#ifdef __cplusplus
	extern "C"
	{
#endif
	#include "VFAlarms.h"
#ifdef __cplusplus
	};
#endif

plcbit vfAlarmPersistentId(struct vfAlarms_Component_typ* alarmComponent, struct vfAlarms_Instance_type* alarm, plcbit AlarmConditionActive, unsigned long* id ){
	// This routine is valid for Persistent alarms only!

	if ( *id == 0) {
		if (AlarmConditionActive) {
			// Set the alarm and return the instance ID of the alarm to be used in MpAlarmXResetID
			*id = MpAlarmXSet( &alarmComponent->link, alarm->_);
		}
	}
	else{
		if ( !AlarmConditionActive ) {
			// Reset the alarm by instance ID.
			MpAlarmXResetID( &alarmComponent->link, *id );
			*id = 0;
		}
	}

	return AlarmConditionActive;

}

plcbit vfAlarmPersistent(struct vfAlarms_Component_typ* alarmComponent, struct vfAlarms_Instance_type* alarm, plcbit AlarmConditionActive){

	return vfAlarmPersistentId( alarmComponent, alarm, AlarmConditionActive, &alarm->id );

}
plcbit vfAlarmPersistentSnippet(struct vfAlarms_Component_typ* alarmComponent, struct vfAlarms_Instance_type* alarm, plcbit AlarmConditionActive, plcstring* snippet){

	if(AlarmConditionActive){
		strncpy(alarm->snippet, snippet, sizeof(alarm->snippet) );
	}
	return vfAlarmPersistentId( alarmComponent, alarm, AlarmConditionActive, &alarm->id );
}

plcbit vfAlarmPersistentSnippetId(struct vfAlarms_Component_typ* alarmComponent, struct vfAlarms_Instance_type* alarm, plcbit AlarmConditionActive, plcstring* snippet, unsigned long* id){

	if(AlarmConditionActive){
		strncpy(alarm->snippet, snippet, sizeof(alarm->snippet) );
	}
	return vfAlarmPersistentId( alarmComponent, alarm, AlarmConditionActive, id);

}
```

### Library Logical/Libraries/VF/VF_COMMON (IEC, version 2.01.0) - 1366 Technologies Miscellaneous Functions
Depends on: standard, MpBase, MpAlarmX, LoopCont, MTData, AsBrStr, astime, LoopConR, AsBrMath

#### RevisionNotes.txt
```
****************************************************************************************************
IMPORTANT: Always update the library version number in the library Properties 'Details' tab.
****************************************************************************************************

Version 2.01 - 1/9/23, W. Stebler
----------------------------------
- VF_Common_MonitoredValue: Added delay to RawValueIsValid input to ensure that disconnected sensors with
  dithering inputs are viewed as invalid.

Version 2.00 - 11/16/22, L. Sullivan
----------------------------------
- Add missing LoopConR lib to dependecy list
- Add AsBrMath lib to dependency list
- Swtich from floor() to brmfloor()
- Switch from strlen() -> brsstrlen() in VF_COMMON_FileNameWithTimestamp
- Rename VF_COMMON_ControlValue_typ and cfg so it doesn't conflict with the VF_COMMON_ControlValue FUB def

Version 1.11 - 12/11/21, W. Stebler
----------------------------------
- Addition of VF_COMMON_DataTypes_enum, VF_COMMON_DatabaseValueCfg_typ, and VF_COMMON_DatabaseValue_typ
  in support of machine data collection.

Version 1.10 - 10/25/21, W. Stebler
----------------------------------
- VF_COMMON_MpAlarmXToggle: Corrected a major bug in the logic of this function that would allow
  alarms to disappear from the alarm list after being acknowledged even if the condition was still active.
  This only occured in instances where the alarm was set up to support multiple instances.

Version 1.09 - 8/22/21, W. Stebler
----------------------------------
- VF_COMMON_ControlValueCfg_typ and VF_COMMON_MonitoredValueCfg_typ now contain DB_Name[] and DisplayName[] properties;
  DB_Name[] replaces the original Name[] peroperty.  DB_CrossReference replaces oroginal PDB_CrossReference.

Version 1.08 - 6/23/21, W. Stebler
----------------------------------
- Added FileNameWithTimestamp function block which returns a filename with timestamp suffix.

Version 1.07 - 4/12/21, W. Stebler
----------------------------------
- Added ControlValue and MonitorValue function blocks.
- Added MTData and LoopCont libraries as dependencies required by these two new functions.

Version 1.06 - 1/29/21, W. Stebler
----------------------------------
- Improved function block comments.
- Added library dependencies required to support MpAlarmX.
- Moved MpAlarmXToggle and CheckAtPosition functions from original location in VF_UTIL library.
- CheckAtPosition renamed to IsValueInRange as this is more generally useful for comparisons.

Version 1.05 - 1/18/21, W. Stebler
----------------------------------
- Removed obsolete CalibratePixelPower function block.

Version 1.04 - 11/16/20, W. Stebler
----------------------------------
- Added function ConvertToHex which converts a UDINT value to its equivalent hexidecimal string.
	You'd think this capabilty would exist in one of the B&R libraries, but I coudn't find it.

Version 1.03 - 10/6/20, W. Stebler
----------------------------------
- Added explicit conversions to REAL data type in CalibratePixelPower (to avoid compiler warning messages).

Version 1.02 - 10/1/20, W. Stebler
----------------------------------
- Added function TON_ScanMicrosec which implements the TON function but wiht a minimum resolution of
	the calling task scan time, rather than the 10msec minimum imposed by the B&R TON function block.
- Added function PulseTrainHiRes which uses the above function to produce pulse trains with ON/OFF resolution
	of the calling task scan time.
- PulseTrainHiRes time Delay, ON, OFF parameters have been changed back to milliseconds and are converted
	internally to microseconds.

Version 1.01 - 8/27/20, R. Singh
----------------------------------
- Added VF_COMMON_CalibratePixelPower function. It uses 2nd order polynomial equation to calibrate power setpoint of every pixel in laser array

Version 1.00 - 8/25/20, W. Stebler
----------------------------------
- Original version.  The PulseTrain function block was relocated from VF_UTIL library to this generic library.
```

#### VF_COMMON.typ - Exported data types
```iecst
TYPE
	LED_Colors :
		( (*Colors associated with status indicator LEDs*)
		LED_OFF,
		LED_Green,
		LED_Yellow,
		LED_Red,
		LED_Blue,
		LED_Gray
		);
	VF_COMMON_LinearScale_typ : 	STRUCT  (*Linear scale factor (raw=PLC units, engineering=user units)*)
		RawMax : INT; (*Max raw units*)
		RawMin : INT; (*Min raw units*)
		RawOffset : INT; (*Optional offset applied to raw value reading prior to scaling*)
		EngineeringMax : REAL; (*Max engineering units*)
		EngineeringMin : REAL; (*Min engineering units*)
		EngineeringUnits : STRING[8]; (*Engineering units descripton (e.g. 'kPa', 'degC', etc.)*)
		DecimalPlaces : USINT; (*Engineering value display decimal places*)
	END_STRUCT;
	VF_COMMON_Constraints_typ : 	STRUCT  (*Constraints used to further limit value entry to a reasonable range for the process*)
		EnableConstraints : BOOL; (*TRUE to enable constraints; FALSE to ignore these values*)
		ScaledMax : REAL; (*Max permitted value in engineering units (typically less than .Scale.EngineeringMax)*)
		ScaledMin : REAL; (*Min permitted value in engineering units (typically greater than .Scale.EngineeringMin)*)
	END_STRUCT;
	VF_COMMON_Limit_typ : 	STRUCT  (*Defines an alarm or warning limit value along with a hysteresis range surrounding it*)
		EnableLimit : BOOL; (*TRUE to enable the limit; FALSE to disable*)
		ScaledValue : REAL; (*The limit value in engineering units*)
		ScaledHysteresis : REAL; (*The hysteresis range that straddles the limit value (1/2 on either side)*)
	END_STRUCT;
	VF_COMMON_LimitConfig_typ : 	STRUCT  (*Limit definition for alarms and warnings*)
		UpperAlarm : VF_COMMON_Limit_typ;
		UpperWarning : VF_COMMON_Limit_typ;
		LowerWarning : VF_COMMON_Limit_typ;
		LowerAlarm : VF_COMMON_Limit_typ;
		DelayAlarm_msec : UINT; (*Time delay (msec) until alarm condition causes an alarm output (set to 0 for no delay)*)
		DelayWarning_msec : UINT; (*Time delay (msec) until warning condition causes an warning output (set to 0 for no delay)*)
		MaxValidRawValue : INT; (*Maximum valid raw value beyond which the OverRange status is turned ON*)
		MinValidRawValue : INT; (*Minimum valid raw value below which the UnderRange status is turned ON*)
		EnableOutOfRange : BOOL; (*TRUE to enable out of range detection; FALSE to disable*)
		DelayOutOfRange_msec : UINT; (*Time delay (msec) until an out of range condition causes an out of range output (set to 0 for no delay)*)
	END_STRUCT;
	VF_COMMON_LimitStatus : 	STRUCT  (*Status of value including alarms and warnings (if configured)*)
		OverRange : BOOL;
		UpperAlarmTripped : BOOL;
		UpperWarningTripped : BOOL;
		LowerWarningTripped : BOOL;
		LowerAlarmTripped : BOOL;
		UnderRange : BOOL;
	END_STRUCT;
	VF_COMMON_MonitoredValueCfg_typ : 	STRUCT  (*Input to the VF_COMMON_MonitoredValue function block*)
		Used : BOOL; (*Set to TRUE if the value is used in code; FALSE to disable (possibly for version-specific reasons)*)
		DB_CrossReference : UINT; (*Cross-reference integer value used by production database to identify this value*)
		DB_Name : STRING[32]; (*Cross-reference string value used by production database to identify this value*)
		DisplayName : STRING[40]; (*Display name of the monitored value*)
		UpdateConfiguration : BOOL; (*Set to TRUE to accept the new configuration; PLC sets to FALSE when new configuration applied*)
		MovingWindowLength : UDINT; (*Number of samples to average (0=disable averaging); use caution when changing at runtime!*)
		Scale : VF_COMMON_LinearScale_typ;
		Limits : VF_COMMON_LimitConfig_typ;
	END_STRUCT;
	VF_COMMON_MonitoredValue_typ : 	STRUCT  (*Input to the VF_COMMON_MonitorValue function block*)
		Disabled : BOOL; (*TRUE if the monitored value is disabled*)
		DB_Name : STRING[32]; (*Cross-reference string value used by production database to identify this value*)
		RawValue : INT; (*Input raw value to be scaled and monitored (typically received from an analog input)*)
		ScaledValue : REAL; (*Scaled engineering value (scaled by the PLC using the linear scaling defined in .Config.Scale), averaged by .MovingAverageSamples number of scans*)
		ScaledValue_NonAveraged : REAL; (*Scaled engineering value (scaled by the PLC using the linear scaling defined in .Config.Scale)*)
		ValueIsValid : BOOL; (*TRUE if the value is currently valid*)
		AlarmsInhibited : BOOL; (*Reflects the current state of the InhibitAlarms input*)
		Status : VF_COMMON_LimitStatus; (*Status of value including alarms and warnings (if configured)*)
		LEDState : USINT; (*LED color associated with the current status of the monitored value*)
		Statistics : MTDataStatistics; (*Statistics calculations based on the scaled value (only active if .MovingWindowLength > 0)*)
		Overflow : BOOL;
		Underflow : BOOL;
		AnalogBad : BOOL;
	END_STRUCT;
	VF_COMMON_ControlledValueCfg_typ : 	STRUCT  (*Input to the VF_COMMON_ControlValue function block*)
		Used : BOOL; (*Set to TRUE if the value is used in code; FALSE to disable (possibly for version-specific reasons)*)
		DB_CrossReference : UINT; (*Cross-reference integer value used by production database to identify this value*)
		DB_Name : STRING[32]; (*Cross-reference string value used by production database to identify this value*)
		DisplayName : STRING[40]; (*Display name of the controlled value*)
		UpdateConfiguration : BOOL; (*Set to TRUE to accept the new configuration; PLC sets to FALSE when new configuration applied*)
		Scale : VF_COMMON_LinearScale_typ;
		Constraints : VF_COMMON_Constraints_typ; (*If constraints are enabled, the InputScaledValue is constrained to withing these limits*)
	END_STRUCT;
	VF_COMMON_ControlledValue_typ : 	STRUCT  (*Input to the VF_COMMON_ControlValue function block*)
		Disabled : BOOL; (*TRUE if the controlled value is disabled*)
		DB_Name : STRING[32]; (*Cross-reference string value used by production database to identify this value*)
		InputScaledValue : REAL; (*Scaled engineering value to be (optionally constrained and) reverse scaled to the output raw value*)
		ScaledValueConstrained : REAL; (*Scaled engineering value after being optionally contstrained*)
		RawValue : INT; (*Output raw value typically sent to an analog output*)
	END_STRUCT;
	VF_COMMON_DBDataTypes_enum :
		( (*Data types supported by machine data collection system.*)
		DT_BOOL_SQL_BIT, (*Store as SQL server 'bit' data type (0, 1) [packed into bytes]*)
		DT_USINT_SQL_TINYINT, (*Store as SQL server 'tinyint' (one byte, unsigned) (0..255)*)
		DT_INT_SQL_SMALLINT, (*Store as SQL server 'smallint' data type (2 bytes) (-32768..32767)*)
		DT_UINT_SQL_INT, (*Store as SQL server 'int' data type (4 bytes) (-2147483648..2147483647)*)
		DT_DINT_SQL_INT, (*Store as SQL server 'int' data type (4 bytes) (-2147483648..2147483647)*)
		DT_UDINT_SQL_BIGINT, (*Store as SQL server 'bigint' data type (8 bytes)*)
		DT_REAL_SQL_REAL, (*Store as SQL server 'real' data type (4 bytes) (3.4E+38)*)
		DT_LREAL_SQL_FLOAT (*Store as SQL server 'float' data type (4/8 bytes) (1.79E+308)*)
		);
	VF_COMMON_DatabaseValueCfg_typ : 	STRUCT  (*Data collection system value configuration*)
		Used : BOOL; (*Set to TRUE if the value is used in code; FALSE to disable (possibly for version-specific reasons)*)
		DB_CrossReference : UINT; (*Cross-reference integer value used by production database to identify this value*)
		DB_Name : STRING[32]; (*Cross-reference string value used by production database to identify this value*)
		DisplayName : STRING[50]; (*Display name of the controlled value*)
		EngineeringUnits : STRING[8]; (*Engineering units descripton (e.g. 'kPa', 'degC', etc.)*)
		DataType : VF_COMMON_DBDataTypes_enum;
		DecimalPlaces : USINT; (*Engineering value display decimal places*)
	END_STRUCT;
	VF_COMMON_DatabaseValue_typ : 	STRUCT  (*Data collection system value*)
		Disabled : BOOL; (*TRUE if the controlled value is disabled*)
		DB_Name : STRING[32]; (*Cross-reference string value used by production database to identify this value*)
		Value : REAL; (*Scaled engineering value to be (optionally constrained and) reverse scaled to the output raw value*)
	END_STRUCT;
END_TYPE
```

#### VF_COMMON.fun - Exported functions and function blocks
```iecst
FUNCTION_BLOCK VF_COMMON_TON_ScanMicrosec (*Timer with a resolution of the calling task scan time*)
	VAR_INPUT
		IN : BOOL := FALSE; (*Set to enable the pulse train, reset to disable/reset*)
		ScanTimeMicrosec : UDINT := 2000; (*PLC task scan time*)
		PT : UDINT := 2000; (*Preset time (microseconds)*)
	END_VAR
	VAR_OUTPUT
		ET : UDINT := 2000; (*Elapsed time (microseconds)*)
		Q : BOOL := FALSE; (*TRUE when the timer is done*)
	END_VAR
	VAR
		scanCountTarget : UDINT := 0;
		scanCount : UDINT := 0;
		enabled : BOOL := FALSE;
	END_VAR
END_FUNCTION_BLOCK

FUNCTION_BLOCK VF_COMMON_PulseTrain (*Generates a pulse train with a resolution of 10 msec*)
	VAR_INPUT
		Enable : BOOL := FALSE; (*Set to enable the pulse train, reset to disable/reset*)
		StartDelay : UDINT := 0; (*Delay (msec) to the start of the pulse train*)
		PulseOnTime : UDINT := 100; (*Pulse ON time (msec)*)
		PulseOffTime : UDINT := 100; (*Pulse OFF time (msec)*)
		NumPulses : UINT := 0; (*Number of pulses to produce (0=infinite)*)
	END_VAR
	VAR_OUTPUT
		NumPulsesCompleted : UINT := 0; (*Number of pulses completed so far (unless NumPulses=0)*)
		Done : BOOL := FALSE; (*TRUE when requested number of pulses has been completed (unless NumPulses=0)*)
		PulseOutput : BOOL := FALSE; (*Pulse output variable*)
		PulseOutputOneScan : BOOL := FALSE; (*Pulse output variable (TRUE for only one scan per pulse)*)
	END_VAR
	VAR
		TON_StartDelay : TON := (0);
		TON_OnState : TON := (0);
		TON_OffState : TON := (0);
		CTU_PulseCounter : CTU;
		startedPulses : BOOL := FALSE;
		pulseHistory : BOOL := FALSE;
		enabled : BOOL := FALSE;
	END_VAR
END_FUNCTION_BLOCK

FUNCTION_BLOCK VF_COMMON_PulseTrainHiRes (*Generates a pulse train with a resolution of the calling task scan time*)
	VAR_INPUT
		Enable : BOOL := FALSE; (*Set to enable the pulse train, reset to disable/reset*)
		ScanTimeMicrosec : UDINT := 2000; (*PLC task scan time (microseconds)*)
		StartDelay : UDINT := 0; (*Delay (msec) to the start of the pulse train*)
		PulseOnTime : UDINT := 100; (*Pulse ON time (msec)*)
		PulseOffTime : UDINT := 100; (*Pulse OFF time (msec)*)
		NumPulses : UINT := 0; (*Number of pulses to produce (0=infinite)*)
	END_VAR
	VAR_OUTPUT
		NumPulsesCompleted : UINT := 0; (*Number of pulses completed so far (unless NumPulses=0)*)
		Done : BOOL := FALSE; (*TRUE when requested number of pulses has been completed (unless NumPulses=0)*)
		PulseOutput : BOOL := FALSE; (*Pulse output variable*)
		PulseOutputOneScan : BOOL := FALSE; (*Pulse output variable (TRUE for only one scan per pulse)*)
	END_VAR
	VAR
		TON_StartDelay : VF_COMMON_TON_ScanMicrosec;
		TON_OnState : VF_COMMON_TON_ScanMicrosec;
		TON_OffState : VF_COMMON_TON_ScanMicrosec;
		CTU_PulseCounter : CTU;
		startedPulses : BOOL := FALSE;
		pulseHistory : BOOL := FALSE;
		enabled : BOOL := FALSE;
	END_VAR
END_FUNCTION_BLOCK

FUNCTION VF_COMMON_ConvertToHex : BOOL (*Converts an unsigned integer value to a hexidecimal string*) (*$GROUP=User,$CAT=User,$GROUPICON=User.png,$CATICON=User.png*)
	VAR_INPUT
		valueToConvert : UDINT;
	END_VAR
	VAR_IN_OUT
		outputHexString : STRING[20];
	END_VAR
	VAR
		quotient : UDINT;
		remainder : UDINT;
		digitIndex : USINT;
	END_VAR
	VAR CONSTANT
		hexDigits : ARRAY[0..15] OF STRING[1] := ['0','1','2','3','4','5','6','7','8','9','A','B','C','D','E','F'];
	END_VAR
END_FUNCTION

FUNCTION VF_COMMON_IsValueInRange : BOOL (*Returns TRUE if specified position is within a defined tolerance band*)
	VAR_INPUT
		TargetValue : LREAL;
		Tolerance : REAL;
		ValueToCompare : LREAL;
	END_VAR
END_FUNCTION

FUNCTION VF_COMMON_MpAlarmXToggle : BOOL (*Sets or resets a named alarm based on CurrentState and InstanceID*)
	VAR_INPUT
		MpLink : MpComIdentType;
		Name : STRING[255];
		AlarmConditionActive : BOOL;
	END_VAR
	VAR_IN_OUT
		InstanceID : UDINT;
	END_VAR
END_FUNCTION

FUNCTION_BLOCK VF_COMMON_ControlValue (*Convert a scaled input value to a raw value (INT)*)
	VAR_INPUT
		Enable : BOOL := FALSE;
		pValueConfig : REFERENCE TO VF_COMMON_ControlledValueCfg_typ; (*Pointer to the controlled value configuration structure*)
		pValue : REFERENCE TO VF_COMMON_ControlledValue_typ; (*Pointer to the controlled value structure*)
	END_VAR
	VAR_OUTPUT
		InternalErrorCode : UINT; (*Error code from internal function blocks, or 0 for no error*)
	END_VAR
	VAR
		fbLCRLimitScale : LCRLimScal;
		initialized : BOOL := FALSE;
		updateConfigComplete : BOOL := FALSE;
		tempScaledValue : REAL;
		lastRawValue : INT := 0;
	END_VAR
END_FUNCTION_BLOCK

FUNCTION_BLOCK VF_COMMON_MonitorValue (*Convert a raw input value (INT) to a scaled value and monitor it for warning/alarm limits with hysterisis*)
	VAR_INPUT
		Enable : BOOL := FALSE;
		RawValue : INT := 0; (*Raw input value to be monitored*)
		RawValueIsValid : BOOL := FALSE; (*Set to TRUE when the raw input value is a valid signal (i.e. when hardware signal is okay)*)
		InhibitAlarms : BOOL := FALSE; (*Set to TRUE to temporarily disable all limit checks (warning, alarm, and out of range)*)
		pValueConfig : REFERENCE TO VF_COMMON_MonitoredValueCfg_typ; (*Pointer to the monitored value configuration structure*)
		pValue : REFERENCE TO VF_COMMON_MonitoredValue_typ; (*Pointer to the monitored value structure*)
	END_VAR
	VAR_OUTPUT
		InternalErrorCode : UINT; (*Error code from internal function blocks, or 0 for no error*)
	END_VAR
	VAR
		fbLCRLimitScale : LCRLimScal;
		fbLC3PointHysteresisAlarm : LC3PHy;
		fbLC3PointHysteresisWarning : LC3PHy;
		fbTONRawValueValid : TON;
		initialized : BOOL := FALSE;
		scaledZero : REAL;
		enableStatistics : BOOL;
		minValidRaw : INT;
		maxValidRaw : INT;
		enOutOfRange : BOOL := FALSE;
		haveOver : BOOL := FALSE;
		haveUnder : BOOL := FALSE;
		enUpperAlarm : BOOL := FALSE;
		enUpperWarn : BOOL := FALSE;
		enLowerWarn : BOOL := FALSE;
		enLowerAlarm : BOOL := FALSE;
		haveUpperAlarm : BOOL := FALSE;
		haveUpperWarn : BOOL := FALSE;
		haveLowerWarn : BOOL := FALSE;
		haveLowerAlarm : BOOL := FALSE;
		outOfRangeDelay : UINT := 0;
		alarmDelay : UINT := 0;
		warningDelay : UINT := 0;
		TON_OutOfRangeDelay : TON;
		TON_AlarmDelay : TON;
		TON_WarningDelay : TON;
		errorCode : UINT;
		lastRawValue : INT := 0;
		lastScaledValue : REAL := 0.0;
	END_VAR
END_FUNCTION_BLOCK

FUNCTION VF_COMMON_FileNameWithTimestamp : BOOL
	VAR_INPUT
		BaseFileName : STRING[100];
		FileExtension : STRING[10];
		CurrentDateAndTime : DATE_AND_TIME;
		IncludeTime : BOOL;
	END_VAR
	VAR_IN_OUT
		OutputFileName : STRING[150];
	END_VAR
	VAR
		dateTimeStruct : DTStructure;
		timeYEAR : STRING[4];
		timeMONTH : STRING[4];
		timeDAY : STRING[4];
		timeHOUR : STRING[4];
		timeMIN : STRING[4];
		timeSEC : STRING[4];
	END_VAR
END_FUNCTION
```

#### VF_COMMON_TON_ScanMicrosec.st - Timer with a resolution of the calling task scan time
```iecst
// ---------------------------------------------------------------------------
// This function block implments a timer with an similar interface to the
// TON function block but with a resolution that matches the scan time of
// the task from which it is called (specifed by ScanTimeMicrosec).
// ---------------------------------------------------------------------------
FUNCTION_BLOCK VF_COMMON_TON_ScanMicrosec

	IF (IN AND enabled) THEN
		scanCount := scanCount + 1;
		ET := scanCount * ScanTimeMicrosec;
		IF (scanCount >= scanCountTarget) THEN
			Q := TRUE;
			scanCount := scanCount - 1;
		END_IF
	ELSE
		enabled := FALSE;
		Q := FALSE;
		ET := 0;
		scanCount := 0;
	END_IF

	// Wait for leading edge of the enable signal.
	IF (IN AND NOT enabled) THEN
		enabled := TRUE;
		Q := FALSE;
		ET := 0;
		// Scan count target is rounded down to the nearest integer value.
		IF (ScanTimeMicrosec <= 0) THEN
			ScanTimeMicrosec := 2000;
		END_IF
		scanCountTarget := REAL_TO_UDINT(brmfloor(UDINT_TO_REAL(PT) / UDINT_TO_REAL(ScanTimeMicrosec)));
	END_IF

END_FUNCTION_BLOCK
```

#### VF_COMMON_PulseTrain.st - Generates a pulse train with a resolution of 10 msec
```iecst
// ---------------------------------------------------------------------------
// This function block generates a pulse train of one or more pulses with an
// optional starting delay. It uses a standard TON function block with a
// 10 msec resolution.
// ---------------------------------------------------------------------------
FUNCTION_BLOCK VF_COMMON_PulseTrain

	IF (Enable AND enabled) THEN

		// If time to start the pulse train...
		IF (StartDelay = 0) OR (TON_StartDelay.Q) THEN

			IF (startedPulses = FALSE) THEN
				PulseOutput := TRUE;
				startedPulses := TRUE;
			END_IF

			// If not done producing pulses...
			IF (NumPulses = 0) OR (CTU_PulseCounter.Q = FALSE) THEN

				IF (TON_OnState.Q) THEN			// on timer is done, turn output OFF
					PulseOutput := FALSE;
					IF (NumPulses > 0) THEN
						CTU_PulseCounter.CU := TRUE;
					END_IF
				END_IF
				IF (TON_OffState.Q) THEN		// off timer is done, turn output ON
					PulseOutput := TRUE;
				END_IF

				IF (PulseOutput = FALSE) THEN	// time the OFF state
					TON_OnState.IN := FALSE;
					TON_OffState.IN := TRUE;
				ELSE 							// time the ON state
					TON_OnState.IN := TRUE;
					TON_OffState.IN := FALSE;
				END_IF

				// Turn on the 'PulseOutputOneScan' output at the start of each pulse.
				PulseOutputOneScan := FALSE;
				IF (PulseOutput) THEN
					IF (NOT pulseHistory) THEN
						pulseHistory := TRUE;
						PulseOutputOneScan := TRUE;
					END_IF
				ELSE
					pulseHistory := FALSE;
				END_IF

			ELSIF (CTU_PulseCounter.Q = TRUE) AND (TON_OffState.Q = TRUE) THEN	// done producing pulses
				Done := TRUE;
			END_IF

		END_IF
	ELSE
		enabled := FALSE;
		startedPulses := FALSE;
		pulseHistory := FALSE;
		TON_StartDelay.IN := FALSE;
		TON_OnState.IN := FALSE;
		TON_OffState.IN := FALSE;
		CTU_PulseCounter.RESET := FALSE;
		PulseOutput := FALSE;
		PulseOutputOneScan := FALSE;
		Done := FALSE;
	END_IF

	// Wait for leading edge, enable start delay, reset internal pulse timers/counter.
	IF (Enable AND NOT enabled) THEN
		enabled := TRUE;
		Done := FALSE;

		IF (StartDelay > 0) THEN
			TON_StartDelay.PT := StartDelay;
			TON_StartDelay.IN := TRUE;
		END_IF

		IF (PulseOnTime < 10) THEN	// minimum 10 msec
			PulseOnTime := 10;
		END_IF
		TON_OnState.PT := PulseOnTime;
		TON_OnState.IN := FALSE;

		IF (PulseOffTime < 10) THEN	// minimum 10 msec
			PulseOffTime := 10;
		END_IF
		TON_OffState.PT := PulseOffTime;
		TON_OffState.IN := FALSE;

		CTU_PulseCounter.PV := NumPulses;
		CTU_PulseCounter.CU := FALSE;
		CTU_PulseCounter.RESET := TRUE;
		startedPulses := FALSE;
	END_IF

	TON_StartDelay();
	TON_OnState();
	TON_OffState();
	CTU_PulseCounter();
	CTU_PulseCounter.CU := FALSE;
	CTU_PulseCounter.RESET := FALSE;
	CTU_PulseCounter();
	NumPulsesCompleted := CTU_PulseCounter.CV;

END_FUNCTION_BLOCK
```

#### VF_COMMON_PulseTrainHiRes.st - Generates a pulse train with a resolution of the calling task scan time
```iecst
// ---------------------------------------------------------------------------
// This function block generates a pulse train of one or more pulses with an
// optional starting delay. It uses a the TON_ScanTimeMicrosec function block
// in this libarary to enable pulse resolution down to the scan time of
// the task from which it is called.
// ---------------------------------------------------------------------------
FUNCTION_BLOCK VF_COMMON_PulseTrainHiRes

	IF (Enable AND enabled) THEN

		TON_StartDelay.ScanTimeMicrosec := ScanTimeMicrosec;
		TON_OnState.ScanTimeMicrosec := ScanTimeMicrosec;
		TON_OffState.ScanTimeMicrosec := ScanTimeMicrosec;

		// If time to start the pulse train...
		IF (StartDelay = 0) OR (TON_StartDelay.Q) THEN

			IF (startedPulses = FALSE) THEN
				PulseOutput := TRUE;
				startedPulses := TRUE;
			END_IF

			// If not done producing pulses...
			IF (NumPulses = 0) OR (CTU_PulseCounter.Q = FALSE) THEN

				IF (TON_OnState.Q) THEN			// on timer is done, turn output OFF
					PulseOutput := FALSE;
					IF (NumPulses > 0) THEN
						CTU_PulseCounter.CU := TRUE;
					END_IF
				END_IF
				IF (TON_OffState.Q) THEN		// off timer is done, turn output ON
					PulseOutput := TRUE;
				END_IF

				IF (PulseOutput = FALSE) THEN	// time the OFF state
					TON_OnState.IN := FALSE;
					TON_OffState.IN := TRUE;
				ELSE 							// time the ON state
					TON_OnState.IN := TRUE;
					TON_OffState.IN := FALSE;
				END_IF

				// Turn on the 'PulseOutputOneScan' output at the start of each pulse.
				PulseOutputOneScan := FALSE;
				IF (PulseOutput) THEN
					IF (NOT pulseHistory) THEN
						pulseHistory := TRUE;
						PulseOutputOneScan := TRUE;
					END_IF
				ELSE
					pulseHistory := FALSE;
				END_IF

			ELSIF (CTU_PulseCounter.Q = TRUE) AND (TON_OffState.Q = TRUE) THEN	// done producing pulses
				Done := TRUE;
			END_IF

		END_IF
	ELSE
		enabled := FALSE;
		startedPulses := FALSE;
		pulseHistory := FALSE;
		TON_StartDelay.IN := FALSE;
		TON_OnState.IN := FALSE;
		TON_OffState.IN := FALSE;
		CTU_PulseCounter.RESET := FALSE;
		PulseOutput := FALSE;
		PulseOutputOneScan := FALSE;
		Done := FALSE;
	END_IF

	// Wait for leading edge, enable start delay, reset internal pulse timers/counter.
	IF (Enable AND NOT enabled) THEN
		enabled := TRUE;
		Done := FALSE;

		IF (StartDelay > 0) THEN
			TON_StartDelay.PT := StartDelay * 1000;
			TON_StartDelay.IN := TRUE;
		END_IF

		TON_OnState.PT := PulseOnTime * 1000;
		TON_OnState.IN := FALSE;

		TON_OffState.PT := PulseOffTime * 1000;
		TON_OffState.IN := FALSE;

		CTU_PulseCounter.PV := NumPulses;
		CTU_PulseCounter.CU := FALSE;
		CTU_PulseCounter.RESET := TRUE;
		startedPulses := FALSE;
	END_IF

	TON_StartDelay();
	TON_OnState();
	TON_OffState();
	CTU_PulseCounter();
	CTU_PulseCounter.CU := FALSE;
	CTU_PulseCounter.RESET := FALSE;
	CTU_PulseCounter();
	NumPulsesCompleted := CTU_PulseCounter.CV;

END_FUNCTION_BLOCK
```

#### VF_COMMON_ConvertToHex.st - Converts an unsigned integer value to a hexidecimal string
```iecst
// ---------------------------------------------------------------------------
// This function block converts an unsigned integer value to a hexidecimal string
// without any prefix/postfix notation.
// ---------------------------------------------------------------------------
FUNCTION VF_COMMON_ConvertToHex

	digitIndex := 7;
	quotient := valueToConvert;
	brsstrcpy(ADR(outputHexString), ADR('00000000'));
	REPEAT
		remainder := quotient MOD 16;
		quotient := quotient / 16;
		brsmemmove(ADR(outputHexString) + digitIndex, ADR(hexDigits[remainder]), 1);
		digitIndex := digitIndex - 1;
	UNTIL
		(quotient <= 0)
	END_REPEAT

	VF_COMMON_ConvertToHex := TRUE;

END_FUNCTION
```

#### VF_COMMON_IsValueInRange.st - Returns TRUE if a specified value is within the range defined by TargetValue +/- Tolerance
```iecst
// ---------------------------------------------------------------------------
// This function returns TRUE if the specified ValueToEvaluate is within the
// range defined by TargetValue +/- Tolerance.
// ---------------------------------------------------------------------------
FUNCTION VF_COMMON_IsValueInRange

	VF_COMMON_IsValueInRange := ((TargetValue - Tolerance) < ValueToCompare) AND (ValueToCompare < (TargetValue + Tolerance));

END_FUNCTION
```

#### VF_COMMON_MpAlarmXToggle.st - Sets or resets a Persistent alarm based on the boolean AlarmState input
```iecst
// ---------------------------------------------------------------------------
// This function sets or resets a persistant alarm based on its current state and instance ID.
// ---------------------------------------------------------------------------
FUNCTION VF_COMMON_MpAlarmXToggle

	// This routine is valid for Persistent alarms only!

	IF (InstanceID = 0) THEN
		IF (AlarmConditionActive) THEN
			// Set the alarm and return the instance ID of the alarm to be used in MpAlarmXResetID
			InstanceID := MpAlarmXSet(MpLink, Name);
		END_IF
	ELSE
		IF (NOT AlarmConditionActive) THEN
			// Reset the alarm by instance ID.
			MpAlarmXResetID(MpLink, InstanceID);
			InstanceID := 0;
		END_IF
	END_IF

	VF_COMMON_MpAlarmXToggle := TRUE;

END_FUNCTION
```

#### VF_COMMON_ControlValue.st - Convert a scaled input value to a raw value (INT) for analog output
```iecst
 (* Convert a scaled input value to a raw value (INT) for analog output *)
FUNCTION_BLOCK VF_COMMON_ControlValue

	IF (Enable) THEN

		// Update configuration on the first pass and on the rising edge of .UpdateConfiguration.
		// This prevents unnecessary code from running once the scaling and limits Convert a scaled input value to a raw value (INT) for analog outputssfare established.
		IF (pValueConfig.UpdateConfiguration AND NOT updateConfigComplete) OR (NOT initialized) THEN

			// Set the linear scale in order to convert from the scaled (engineering) value ot the raw (system) output value.
			fbLCRLimitScale.x1 := pValueConfig.Scale.EngineeringMin;
			fbLCRLimitScale.x2 := pValueConfig.Scale.EngineeringMax;
			fbLCRLimitScale.y1 := INT_TO_REAL(pValueConfig.Scale.RawMin);
			fbLCRLimitScale.y2 := INT_TO_REAL(pValueConfig.Scale.RawMax);

			// If constraints are not enabled, default them to the engineering scale limits.
			// Constraints can only be used to limit the range of values to less than then engineering range.
			IF (NOT pValueConfig.Constraints.EnableConstraints) THEN
				pValueConfig.Constraints.ScaledMax := pValueConfig.Scale.EngineeringMax;
				pValueConfig.Constraints.ScaledMin := pValueConfig.Scale.EngineeringMin;
			END_IF

			initialized := TRUE;
			lastRawValue := 0;

			// Reset the update configuration flag to indicate completion.
			IF (pValueConfig.UpdateConfiguration) THEN
				pValueConfig.UpdateConfiguration := FALSE;
			END_IF
		END_IF

		// Constrain the input value as required.
		tempScaledValue := pValue.InputScaledValue;
		IF (pValueConfig.Constraints.EnableConstraints) THEN
			// When max > min...
			IF (pValueConfig.Constraints.ScaledMax > pValueConfig.Constraints.ScaledMin) THEN
				IF (tempScaledValue > pValueConfig.Constraints.ScaledMax) THEN
					tempScaledValue := pValueConfig.Constraints.ScaledMax;
				ELSIF (tempScaledValue < pValueConfig.Constraints.ScaledMin) THEN
					tempScaledValue := pValueConfig.Constraints.ScaledMin;
				END_IF
			ELSE // when max < min...
				IF (tempScaledValue < pValueConfig.Constraints.ScaledMax) THEN
					tempScaledValue := pValueConfig.Constraints.ScaledMax;
				ELSIF (tempScaledValue > pValueConfig.Constraints.ScaledMin) THEN
					tempScaledValue := pValueConfig.Constraints.ScaledMin;
				END_IF
			END_IF
		END_IF

		pValue.Disabled := FALSE;
		pValue.ScaledValueConstrained := tempScaledValue;

		// Convert the the scaled value to a raw value.
		fbLCRLimitScale(x := tempScaledValue);
		lastRawValue := REAL_TO_INT(fbLCRLimitScale.y);
		pValue.RawValue := lastRawValue;

		InternalErrorCode := 0;

	ELSE

		initialized := FALSE;
		pValue.Disabled := TRUE;
		pValue.ScaledValueConstrained := 0.0;
		pValue.RawValue := lastRawValue;
		InternalErrorCode := 0;

	END_IF

END_FUNCTION_BLOCK
```

#### VF_COMMON_MonitorValue.st - Convert a raw input value (INT) to a scaled value and monitor it for warning/alarm limits
```iecst
 (* Convert a raw input value (INT) to a scaled value and monitor it for warning/alarm limits *)
FUNCTION_BLOCK VF_COMMON_MonitorValue

	IF (Enable) THEN

		// Update configuration on the first pass and on the rising edge of .UpdateConfiguration.
		// This prevents unnecessary code from running once the scaling and limits are established.
		IF (pValueConfig.UpdateConfiguration) OR (NOT initialized) THEN

			// Invert the linear scale in order to convert the alarm limits from scaled (engineering) values to raw (system) values.
			// The raw values are rounded to the nearest integer as required by the LCRLimScal() function block.
			fbLCRLimitScale.x1 := pValueConfig.Scale.EngineeringMin;
			fbLCRLimitScale.x2 := pValueConfig.Scale.EngineeringMax;
			fbLCRLimitScale.y1 := INT_TO_REAL(pValueConfig.Scale.RawMin);
			fbLCRLimitScale.y2 := INT_TO_REAL(pValueConfig.Scale.RawMax);

			// Configure out of range limits.
			maxValidRaw := pValueConfig.Limits.MaxValidRawValue;
			minValidRaw := pValueConfig.Limits.MinValidRawValue;
			enOutOfRange := pValueConfig.Limits.EnableOutOfRange;
			outOfRangeDelay := pValueConfig.Limits.DelayOutOfRange_msec;
			TON_OutOfRangeDelay.PT := REAL_TO_TIME(outOfRangeDelay);
			TON_OutOfRangeDelay.IN := FALSE;

			// Configure ALARM limits, if enabled.
			enLowerAlarm := pValueConfig.Limits.LowerAlarm.EnableLimit;
			enUpperAlarm := pValueConfig.Limits.UpperAlarm.EnableLimit;
			alarmDelay := pValueConfig.Limits.DelayAlarm_msec;
			TON_AlarmDelay.PT := REAL_TO_TIME(alarmDelay);
			TON_AlarmDelay.IN := FALSE;

			// Calculate the raw value representing a scaled value of zero.
			fbLCRLimitScale(x := 0.0);
			scaledZero := fbLCRLimitScale.y;

			fbLC3PointHysteresisAlarm.enable := (enLowerAlarm OR enUpperAlarm);
			IF (enLowerAlarm) THEN
				fbLCRLimitScale(x := pValueConfig.Limits.LowerAlarm.ScaledValue);
				fbLC3PointHysteresisAlarm.xsetvalue1 := REAL_TO_INT(fbLCRLimitScale.y);
				fbLCRLimitScale(x := pValueConfig.Limits.LowerAlarm.ScaledHysteresis);
				fbLC3PointHysteresisAlarm.hysteresis1 := REAL_TO_UINT(fbLCRLimitScale.y - scaledZero);
			ELSE
				fbLC3PointHysteresisAlarm.xsetvalue1 := -32768;
				fbLC3PointHysteresisAlarm.hysteresis1 := 0;
			END_IF
			IF (enUpperAlarm) THEN
				fbLCRLimitScale(x := pValueConfig.Limits.UpperAlarm.ScaledValue);
				fbLC3PointHysteresisAlarm.xsetvalue2 := REAL_TO_INT(fbLCRLimitScale.y);
				fbLCRLimitScale(x := pValueConfig.Limits.UpperAlarm.ScaledHysteresis);
				fbLC3PointHysteresisAlarm.hysteresis2 := REAL_TO_UINT(fbLCRLimitScale.y - scaledZero);
			ELSE
				fbLC3PointHysteresisAlarm.xsetvalue2 := 32767;
				fbLC3PointHysteresisAlarm.hysteresis2 := 0;
			END_IF
			fbLC3PointHysteresisAlarm.ymax := 1;	// above upper limit
			fbLC3PointHysteresisAlarm.ymid := 0;	// within limits
			fbLC3PointHysteresisAlarm.ymin := -1;	// below lower limit
			// Set the starting point midway between the two setpoints.
			fbLC3PointHysteresisAlarm.xstart := fbLC3PointHysteresisAlarm.xsetvalue1 + ((fbLC3PointHysteresisAlarm.xsetvalue2 - fbLC3PointHysteresisAlarm.xsetvalue1) / 2);

			// Configure WARNING limits, if enabled.
			enLowerWarn := pValueConfig.Limits.LowerWarning.EnableLimit;
			enUpperWarn := pValueConfig.Limits.UpperWarning.EnableLimit;
			warningDelay := pValueConfig.Limits.DelayWarning_msec;
			TON_WarningDelay.PT := REAL_TO_TIME(warningDelay);
			TON_WarningDelay.IN := FALSE;

			fbLC3PointHysteresisWarning.enable := (enLowerWarn OR enUpperWarn);
			IF (enLowerWarn) THEN
				fbLCRLimitScale(x := pValueConfig.Limits.LowerWarning.ScaledValue);
				fbLC3PointHysteresisWarning.xsetvalue1 := REAL_TO_INT(fbLCRLimitScale.y);
				fbLCRLimitScale(x :=  pValueConfig.Limits.LowerWarning.ScaledHysteresis);
				fbLC3PointHysteresisWarning.hysteresis1 := REAL_TO_UINT(fbLCRLimitScale.y - scaledZero);
			ELSE
				fbLC3PointHysteresisWarning.xsetvalue1 := -32768;
				fbLC3PointHysteresisWarning.hysteresis1 := 0;
			END_IF
			IF (enUpperWarn) THEN
				fbLCRLimitScale(x := pValueConfig.Limits.UpperWarning.ScaledValue);
				fbLC3PointHysteresisWarning.xsetvalue2 := REAL_TO_INT(fbLCRLimitScale.y);
				fbLCRLimitScale(x := pValueConfig.Limits.UpperWarning.ScaledHysteresis);
				fbLC3PointHysteresisWarning.hysteresis2 := REAL_TO_UINT(fbLCRLimitScale.y - scaledZero);
			ELSE
				fbLC3PointHysteresisWarning.xsetvalue2 := 32767;
				fbLC3PointHysteresisWarning.hysteresis2 := 0;
			END_IF
			fbLC3PointHysteresisWarning.ymax := 1;	// above upper limit
			fbLC3PointHysteresisWarning.ymid := 0;	// within limits
			fbLC3PointHysteresisWarning.ymin := -1;	// below lower limit
			// Set the starting point midway between the two setpoints.
			fbLC3PointHysteresisWarning.xstart := fbLC3PointHysteresisWarning.xsetvalue1 + ((fbLC3PointHysteresisWarning.xsetvalue2 - fbLC3PointHysteresisWarning.xsetvalue1) / 2);

			// Set the linear scale in order to conver the raw (system) input value to a scaled (engineering) output value.
			fbLCRLimitScale.x1 := INT_TO_REAL(pValueConfig.Scale.RawMin);
			fbLCRLimitScale.x2 := INT_TO_REAL(pValueConfig.Scale.RawMax);
			fbLCRLimitScale.y1 := pValueConfig.Scale.EngineeringMin;
			fbLCRLimitScale.y2 := pValueConfig.Scale.EngineeringMax;

			// Set up the moving window size.
			IF (pValueConfig.MovingWindowLength > 0) THEN
				enableStatistics := TRUE;
				pValue.Statistics.Reset := TRUE;
				pValue.Statistics();
				pValue.Statistics.MovingWindowLength := pValueConfig.MovingWindowLength;
				pValue.Statistics.Enable := TRUE;
				pValue.Statistics();
			ELSE
				enableStatistics := FALSE;
				pValue.Statistics.Enable := FALSE;
				pValue.Statistics();
			END_IF

			initialized := TRUE;
			lastRawValue := 0;
			lastScaledValue := 0.0;

			// Reset the update configuration flag to indicate completion.
			IF (pValueConfig.UpdateConfiguration) THEN
				pValueConfig.UpdateConfiguration := FALSE;
			END_IF
		END_IF

		// Update the value structure with the input raw value and its status.
		pValue.Disabled := FALSE;
		pValue.RawValue := RawValue;
		// Fixed 2 second delay to prevent disconnected sensor with dithering IO status bits (e.g. underflow/overflow) from participating the scaling code.
		fbTONRawValueValid.IN := RawValueIsValid;
		fbTONRawValueValid.PT := T#20ms;
		pValue.ValueIsValid := fbTONRawValueValid.Q;

		// If the raw value is valid, monitor the alarm and warning conditions with hysterisis;
		// otheriwse, the output value remains at its last valid value and the alarm/warning outputs are set to FALSE.
		IF (fbTONRawValueValid.Q) THEN

			// Capture the raw value, adjusted by any specified raw offset.
			lastRawValue := RawValue + pValueConfig.Scale.RawOffset;

			// Convert the raw value to a scaled value.
			fbLCRLimitScale(x := lastRawValue);
			pValue.ScaledValue_NonAveraged := fbLCRLimitScale.y;
			lastScaledValue := pValue.ScaledValue_NonAveraged;

			// If statistics are enabled, add the value and recompute staticstics.
			IF (enableStatistics) THEN
				pValue.Statistics.In := lastScaledValue;
				pValue.Statistics();
				pValue.ScaledValue := pValue.Statistics.Mean;
			ELSE
				pValue.ScaledValue := lastScaledValue;
			END_IF

			// If the raw value is on or outside of the limits, flag the out of range condition.
			IF (enOutOfRange) AND (NOT InhibitAlarms) THEN
				haveOver := (lastRawValue >= maxValidRaw);
				haveUnder := (lastRawValue <= minValidRaw);
				// Delay the range output if a non-zero time (in msec) was specified.
				IF (outOfRangeDelay > 0) THEN
					TON_OutOfRangeDelay.IN := (haveUnder OR haveOver);
					pValue.Status.OverRange := (TON_OutOfRangeDelay.Q AND haveOver);
					pValue.Status.UnderRange := (TON_OutOfRangeDelay.Q AND haveUnder);
				ELSE
					TON_OutOfRangeDelay.IN := FALSE;
					pValue.Status.OverRange := haveOver;
					pValue.Status.UnderRange := haveUnder;
				END_IF
			ELSE
				pValue.Status.OverRange := FALSE;
				pValue.Status.UnderRange := FALSE;
			END_IF

			InternalErrorCode := 0;

			// Check for ALARM conditions based on input value (LC3PHy() function block takes care of hysteresis).
			// Error code (if any) from the LC3PHy function blocks are reported on the InternalErrorCode output.
			fbLC3PointHysteresisAlarm(x := lastRawValue);
			IF (NOT InhibitAlarms) THEN
				errorCode := fbLC3PointHysteresisAlarm.status;
				IF (errorCode <> 0) AND (enLowerAlarm OR enUpperAlarm) THEN
					InternalErrorCode := errorCode;
					pValue.Status.UpperAlarmTripped := TRUE;
					pValue.Status.LowerAlarmTripped := TRUE;
				ELSE
					haveUpperAlarm := SEL(enUpperAlarm, FALSE, fbLC3PointHysteresisAlarm.ymx);
					haveLowerAlarm := SEL(enLowerAlarm, FALSE, fbLC3PointHysteresisAlarm.ymn);
					// Delay the alarm output if a non-zero time (in msec) was specified.
					IF (alarmDelay > 0) THEN
						TON_AlarmDelay.IN := (haveUpperAlarm OR haveLowerAlarm);
						pValue.Status.UpperAlarmTripped := (TON_AlarmDelay.Q AND haveUpperAlarm);
						pValue.Status.LowerAlarmTripped := (TON_AlarmDelay.Q AND haveLowerAlarm);
					ELSE
						TON_AlarmDelay.IN := FALSE;
						pValue.Status.UpperAlarmTripped := haveUpperAlarm;
						pValue.Status.LowerAlarmTripped := haveLowerAlarm;
					END_IF
				END_IF
			ELSE
				pValue.Status.UpperAlarmTripped := FALSE;
				pValue.Status.LowerAlarmTripped := FALSE;
			END_IF

			// Check for WARNING conditions based on input value (LC3PHy() function block takes care of hysteresis).
			fbLC3PointHysteresisWarning(x := lastRawValue);
			IF (NOT InhibitAlarms) THEN
				errorCode := fbLC3PointHysteresisWarning.status;
				IF (errorCode <> 0) AND (enLowerWarn OR enUpperWarn) THEN
					IF (InternalErrorCode = 0) THEN  // only set error code if it was not already set above
						InternalErrorCode := errorCode;
					END_IF
					pValue.Status.UpperWarningTripped := TRUE;
					pValue.Status.LowerWarningTripped := TRUE;
				ELSE
					haveUpperWarn := SEL(enUpperWarn, FALSE, fbLC3PointHysteresisWarning.ymx);
					haveLowerWarn := SEL(enLowerWarn, FALSE, fbLC3PointHysteresisWarning.ymn);
					// Delay the warning output if a non-zero time (in msec) was specified.
					IF (warningDelay > 0) THEN
						TON_WarningDelay.IN := (haveUpperWarn OR haveLowerWarn);
						pValue.Status.UpperWarningTripped := (TON_WarningDelay.Q AND haveUpperWarn);
						pValue.Status.LowerWarningTripped := (TON_WarningDelay.Q AND haveLowerWarn);
					ELSE
						TON_WarningDelay.IN := FALSE;
						pValue.Status.UpperWarningTripped := haveUpperWarn;
						pValue.Status.LowerWarningTripped := haveLowerWarn;
					END_IF
				END_IF
			ELSE
				pValue.Status.UpperWarningTripped := FALSE;
				pValue.Status.LowerWarningTripped := FALSE;
			END_IF

			pValue.AlarmsInhibited := InhibitAlarms;

			// Set Status LED color based on current status.
			IF (InhibitAlarms) THEN
				pValue.LEDState := DINT_TO_USINT(LED_Gray);
			ELSIF (pValue.Status.OverRange OR pValue.Status.UnderRange) THEN
				pValue.LEDState := DINT_TO_USINT(LED_Blue);
			ELSIF (pValue.Status.LowerAlarmTripped OR pValue.Status.UpperAlarmTripped) THEN
				pValue.LEDState := DINT_TO_USINT(LED_Red);
			ELSIF (pValue.Status.LowerWarningTripped OR pValue.Status.UpperWarningTripped) THEN
				pValue.LEDState := DINT_TO_USINT(LED_Yellow);
			ELSE
				pValue.LEDState := DINT_TO_USINT(LED_Green);
			END_IF

		ELSE  // IF (RawValueIsValid)

			pValue.ScaledValue := lastScaledValue;
			pValue.ScaledValue_NonAveraged := lastScaledValue;
			pValue.AlarmsInhibited := InhibitAlarms;
			pValue.Status.OverRange := NOT InhibitAlarms;
			pValue.Status.UnderRange := NOT InhibitAlarms;
			pValue.Status.UpperAlarmTripped := FALSE;
			pValue.Status.UpperWarningTripped := FALSE;
			pValue.Status.LowerWarningTripped := FALSE;
			pValue.Status.LowerAlarmTripped := FALSE;
			pValue.LEDState := DINT_TO_USINT(LED_Gray);
			InternalErrorCode := 0;
			TON_OutOfRangeDelay.IN := FALSE;
			TON_AlarmDelay.IN := FALSE;
			TON_WarningDelay.IN := FALSE;
		END_IF

	ELSE  // IF (Enable)

		initialized := FALSE;
		pValue.RawValue := 0;
		pValue.ScaledValue := 0.0;
		pValue.ScaledValue_NonAveraged := 0.0;
		pValue.ValueIsValid := FALSE;
		pValue.Disabled := TRUE;
		pValue.AlarmsInhibited := FALSE;
		pValue.Status.OverRange := FALSE;
		pValue.Status.UnderRange := FALSE;
		pValue.Status.UpperAlarmTripped := FALSE;
		pValue.Status.UpperWarningTripped := FALSE;
		pValue.Status.LowerWarningTripped := FALSE;
		pValue.Status.LowerAlarmTripped := FALSE;
		pValue.LEDState :=  DINT_TO_USINT(LED_OFF);
		InternalErrorCode := 0;
		fbTONRawValueValid.IN := FALSE;
		TON_OutOfRangeDelay.IN := FALSE;
		TON_AlarmDelay.IN := FALSE;
		TON_WarningDelay.IN := FALSE;

	END_IF

	fbTONRawValueValid();
	TON_OutOfRangeDelay();
	TON_AlarmDelay();
	TON_WarningDelay();

END_FUNCTION_BLOCK
```

#### VF_COMMON_FileNameWithTimestamp.st - Converts an unsigned integer value to a hexidecimal string
```iecst
// ---------------------------------------------------------------------------
// This function block appends a timestamp to the specified filename.
// ---------------------------------------------------------------------------
FUNCTION VF_COMMON_FileNameWithTimestamp

	DT_TO_DTStructure(CurrentDateAndTime, ADR(dateTimeStruct));

	// UINT values
	timeYEAR := UINT_TO_STRING(dateTimeStruct.year);
	// USINT values
	timeMONTH := USINT_TO_STRING(dateTimeStruct.month);
	timeDAY := USINT_TO_STRING(dateTimeStruct.day);
	timeHOUR := USINT_TO_STRING(dateTimeStruct.hour);
	timeMIN := USINT_TO_STRING(dateTimeStruct.minute);
	timeSEC := USINT_TO_STRING(dateTimeStruct.second);

	brsstrcpy(ADR(OutputFileName), ADR(BaseFileName));

	brsstrcat(ADR(OutputFileName), ADR('_'));
	brsstrcat(ADR(OutputFileName), ADR(timeYEAR));

	brsstrcat(ADR(OutputFileName), ADR('_'));
	IF (brsstrlen(ADR(timeMONTH)) = 1) THEN
		brsstrcat(ADR(OutputFileName), ADR('0'));
	END_IF
	brsstrcat(ADR(OutputFileName), ADR(timeMONTH));

	brsstrcat(ADR(OutputFileName), ADR('_'));
	IF (brsstrlen(ADR(timeDAY)) = 1) THEN
		brsstrcat(ADR(OutputFileName), ADR('0'));
	END_IF
	brsstrcat(ADR(OutputFileName), ADR(timeDAY));

	IF (IncludeTime) THEN
		brsstrcat(ADR(OutputFileName), ADR('_'));
		IF (brsstrlen(ADR(timeHOUR)) = 1) THEN
			brsstrcat(ADR(OutputFileName), ADR('0'));
		END_IF
		brsstrcat(ADR(OutputFileName), ADR(timeHOUR));

		brsstrcat(ADR(OutputFileName), ADR('_'));
		IF (brsstrlen(ADR(timeMIN)) = 1) THEN
			brsstrcat(ADR(OutputFileName), ADR('0'));
		END_IF
		brsstrcat(ADR(OutputFileName), ADR(timeMIN));

		brsstrcat(ADR(OutputFileName), ADR('_'));
		IF (brsstrlen(ADR(timeSEC)) = 1) THEN
			brsstrcat(ADR(OutputFileName), ADR('0'));
		END_IF
		brsstrcat(ADR(OutputFileName), ADR(timeSEC));
	END_IF

	brsstrcat(ADR(OutputFileName), ADR(FileExtension));

	VF_COMMON_FileNameWithTimestamp := TRUE;

END_FUNCTION
```

### Library Logical/Libraries/VF/ToolBox (ANSIC)

#### ToolBox.fun - Exported functions and function blocks
```iecst
FUNCTION allZero : BOOL
	VAR_INPUT
		pData : UDINT;
		szData : UINT;
	END_VAR
END_FUNCTION

{REDUND_ERROR} FUNCTION EdgePosArray : BOOL (*Trigger edges on an array of booleans*) (*$GROUP=User,$CAT=User,$GROUPICON=User.png,$CATICON=User.png*)
	VAR_INPUT
		Level : REFERENCE TO BOOL;
		PreviousLevel : REFERENCE TO BOOL;
		Edge : REFERENCE TO BOOL;
		Size : UINT;
	END_VAR
END_FUNCTION

{REDUND_ERROR} FUNCTION EdgeNegArray : BOOL (*Trigger edges on an array of booleans*) (*$GROUP=User,$CAT=User,$GROUPICON=User.png,$CATICON=User.png*)
	VAR_INPUT
		Level : REFERENCE TO BOOL;
		PreviousLevel : REFERENCE TO BOOL;
		Edge : REFERENCE TO BOOL;
		Size : UINT;
	END_VAR
END_FUNCTION

{REDUND_ERROR} FUNCTION EdgeArray : BOOL (*Trigger edges on an array of booleans*) (*$GROUP=User,$CAT=User,$GROUPICON=User.png,$CATICON=User.png*)
	VAR_INPUT
		Level : REFERENCE TO BOOL;
		PreviousLevel : REFERENCE TO BOOL;
		Edge : REFERENCE TO BOOL;
		Size : UINT;
	END_VAR
END_FUNCTION
```

#### EdgeArray.c
```c
#include <bur/plctypes.h>
#ifdef __cplusplus
	extern "C"
	{
#endif
	#include "ToolBox.h"
#ifdef __cplusplus
	};
#endif

/* Trigger edges on an array of booleans */
plcbit EdgePosArray(plcbit* Level, plcbit* PreviousLevel, plcbit* Edge, unsigned short Size)
{
	int i;
	for( i=0; i< Size/sizeof(BOOL); i++ ){
		if( Level[i] && !PreviousLevel[i] ){
			Edge[i] = 1;
		}
		PreviousLevel[i] = 	Level[i];
	}
}

/* Trigger edges on an array of booleans */
plcbit EdgeNegArray(plcbit* Level, plcbit* PreviousLevel, plcbit* Edge, unsigned short Size)
{
	int i;
	for( i=0; i< Size/sizeof(BOOL); i++ ){
		if( !Level[i] && PreviousLevel[i] ){
			Edge[i] = 1;
		}
		PreviousLevel[i] = 	Level[i];
	}
}

/* Trigger edges on an array of booleans */
plcbit EdgeArray(plcbit* Level, plcbit* PreviousLevel, plcbit* Edge, unsigned short Size)
{
	int i;
	for( i=0; i< Size/sizeof(BOOL); i++ ){
		if( Level[i] != PreviousLevel[i] ){
			Edge[i] = 1;
		}
		PreviousLevel[i] = 	Level[i];
	}
}
```

#### allZero.c
```c
#include <bur/plctypes.h>
#ifdef __cplusplus
	extern "C"
	{
#endif
	#include "ToolBox.h"
#ifdef __cplusplus
	};
#endif

#include "string.h"

/* Check if all the data is zero */
plcbit allZero( UDINT pData, UINT size )
{
	switch(size){
		case 0: return 1;
		case 1: return  (*(char*)pData == 0);
		default: return (*(char*)pData == 0) && memcmp(pData, pData + 1, size - 1) == 0;
	}
}
```

### Library Logical/Libraries/VF/VFValve (IEC)

#### Types.typ - Exported data types
```iecst
TYPE
	vfValveBasicInternal_typ : 	STRUCT
		valveTimeOutTimer : TON; (*timeout if a command to open or close is sent and it hasnt completed*)
		valveCycleTimer : TON; (*cycle time for a rapid open/close operation*)
		valveState : vfValveBasicStates_typ;
		valveErrorState : vfValveBasicStates_typ;
		actuationDelayTimer : TON;
		oldDoOpen : BOOL;
		oldDoClose : BOOL;
	END_STRUCT;
	vfValveBasicInputs_typ : 	STRUCT
		closeLimitSensor : BOOL;
		openLimitSensor : BOOL;
		adrParameters : REFERENCE TO ValveParameters_typ;
		parameters : ValveParameters_typ;
		adrCommands : REFERENCE TO ValveCommands_typ;
		commands : ValveCommands_typ;
	END_STRUCT;
	vfValveBasicOutputs_typ : 	STRUCT
		OpenValveSignal : BOOL;
		CloseValveSignal : BOOL;
		status : ValveStatus_typ;
	END_STRUCT;
	vfValveBasicStates_typ :
		(
		vfVALVE_BASIC_WAIT_FOR_COMMANDS,
		vfVALVE_BASIC_OPEN,
		vfVALVE_BASIC_CLOSE,
		vfVALVE_BASIC_CYCLE_OPEN,
		vfVALVE_BASIC_CYCLE_CLOSE,
		vfVALVE_BASIC_STOP,
		vfVALVE_BASIC_ERROR
		);
END_TYPE
```

#### ImportedTypes.typ
```iecst
TYPE
	ValveCommands_typ : 	STRUCT
		open : BOOL;
		close : BOOL;
		cycle : BOOL;
		stop : BOOL;
		errReset : BOOL;
	END_STRUCT;
	ValveHandling_typ : 	STRUCT
		commands : ValveCommands_typ;
		parameters : ValveParameters_typ;
		status : ValveStatus_typ;
	END_STRUCT;
	ValveParameters_typ : 	STRUCT
		TimeOutValue : TIME; (*timeout of the valve (not opened or closed despite command)*)
		hasLimitSensors : BOOL; (*FALSE if no limit sensors are used to determine valve position*)
		enabled : BOOL;
		actuationDelay : TIME; (*If option of "no limit" sensors is selected, this is a delay to allow the valve to actuate before reporting on new status*)
		cycleTime : UDINT; (*when cycling this is the amount of time it stays in the open state*)
	END_STRUCT;
	ValveStatus_typ : 	STRUCT
		busy : BOOL;
		opened : BOOL;
		closed : BOOL;
		middle : BOOL;
		cycling : BOOL;
		leftOpened : BOOL;
		leftClosed : BOOL;
		leftMiddle : BOOL;
		rightOpened : BOOL;
		rightClosed : BOOL;
		rightMiddle : BOOL;
		frontLeftOpened : BOOL;
		rearLeftOpened : BOOL;
		frontLeftClosed : BOOL;
		rearLeftClosed : BOOL;
		frontLeftMiddle : BOOL;
		rearLeftMiddle : BOOL;
		frontRightOpened : BOOL;
		rearRightOpened : BOOL;
		frontRightClosed : BOOL;
		rearRightClosed : BOOL;
		frontRightMiddle : BOOL;
		rearRightMiddle : BOOL;
		doOpen : BOOL;
		doClose : BOOL;
		readyForCommand : BOOL;
		safeEnabled : BOOL;
		error : BOOL;
		reachedFullOpen : BOOL;
		fbState : STRING[20];
		actualCycleTimeMsec : UDINT;
	END_STRUCT;
END_TYPE
```

#### VFValve.fun - Exported functions and function blocks
```iecst
FUNCTION_BLOCK vfValveBasic
	VAR_INPUT
		Inputs : vfValveBasicInputs_typ;
	END_VAR
	VAR_OUTPUT
		Outputs : vfValveBasicOutputs_typ;
	END_VAR
	VAR
		pCommandWriteBack : REFERENCE TO ValveCommands_typ;
		internal : vfValveBasicInternal_typ;
	END_VAR
END_FUNCTION_BLOCK
```
